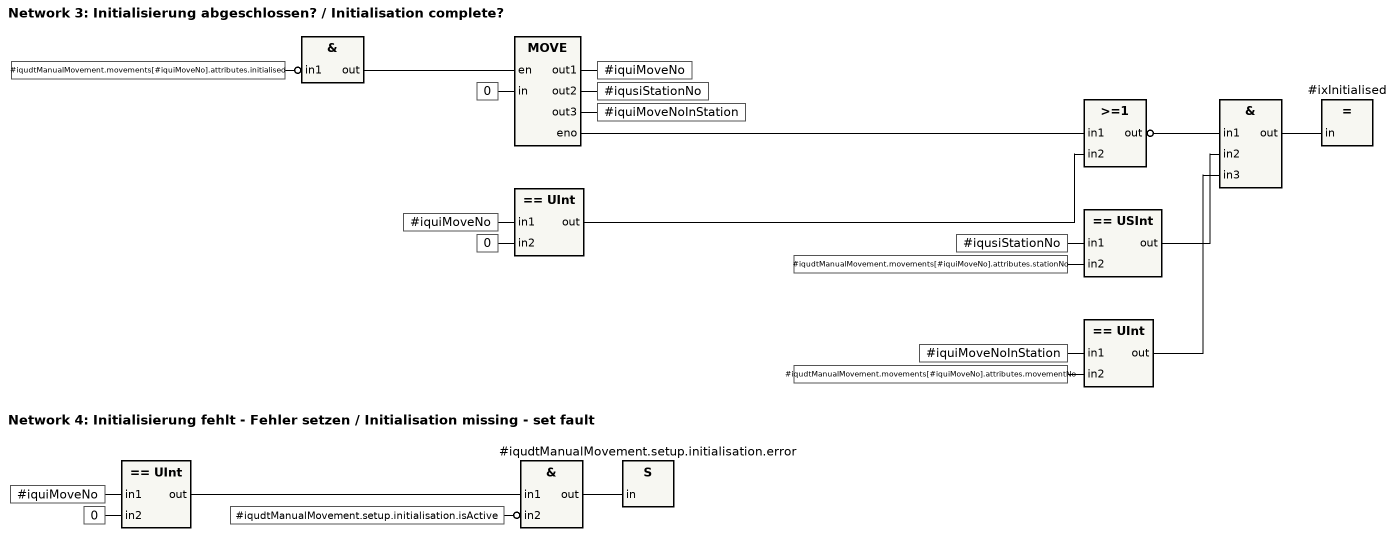
   #_w1 := NOT #iqudtManualMovement.movements[#iquiMoveNo].attributes.initialised;
   IF #_w1 THEN
       #iquiMoveNo := 0;
       #iqusiStationNo := 0;
       #iquiMoveNoInStation := 0;
   END_IF;
   #ixInitialised := NOT (#_w1 OR (#iquiMoveNo = 0)) AND (#iqusiStationNo = #iqudtManualMovement.movements[#iquiMoveNo].attributes.stationNo) AND (#iquiMoveNoInStation = #iqudtManualMovement.movements[#iquiMoveNo].attributes.movementNo);
END_REGION

REGION Network 4: Initialisierung fehlt - Fehler setzen / Initialisation missing - set fault
   IF (#iquiMoveNo = 0) AND NOT #iqudtManualMovement.setup.initialisation.isActive THEN
       #iqudtManualMovement.setup.initialisation.error := TRUE;
   END_IF;
END_REGION

REGION Network 5: Sichtbarkeit / Visibility
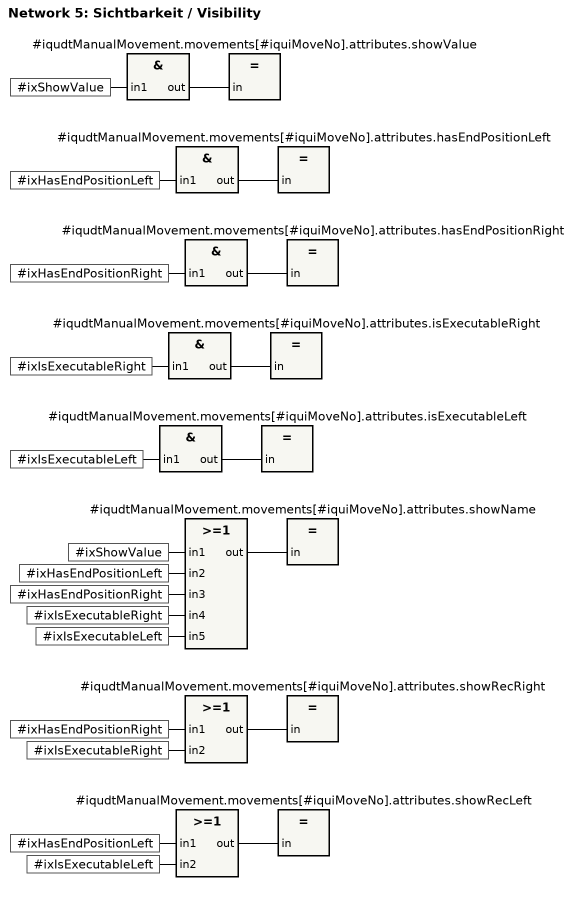
   #iqudtManualMovement.movements[#iquiMoveNo].attributes.showValue := #ixShowValue;
   #iqudtManualMovement.movements[#iquiMoveNo].attributes.hasEndPositionLeft := #ixHasEndPositionLeft;
   #iqudtManualMovement.movements[#iquiMoveNo].attributes.hasEndPositionRight := #ixHasEndPositionRight;
   #iqudtManualMovement.movements[#iquiMoveNo].attributes.isExecutableRight := #ixIsExecutableRight;
   #iqudtManualMovement.movements[#iquiMoveNo].attributes.isExecutableLeft := #ixIsExecutableLeft;
   #iqudtManualMovement.movements[#iquiMoveNo].attributes.showName := #ixShowValue OR #ixHasEndPositionLeft OR #ixHasEndPositionRight OR #ixIsExecutableRight OR #ixIsExecutableLeft;
   #iqudtManualMovement.movements[#iquiMoveNo].attributes.showRecRight := #ixHasEndPositionRight OR #ixIsExecutableRight;
   #iqudtManualMovement.movements[#iquiMoveNo].attributes.showRecLeft := #ixHasEndPositionLeft OR #ixIsExecutableLeft;
END_REGION
END_FUNCTION

FUNCTION "InitManualMovements" : Void   // FC909, SCL
{ S7_Optimized_Access := 'TRUE' }
VERSION : 0.1
   VAR_IN_OUT
      iqarudtMovements : Array[0.."SYS_MANUALMOVEMENTS"] of "typeManualMove";
   END_VAR
   VAR_TEMP
      ttusiCounter : USInt;
   END_VAR
BEGIN
   // Ersteller: Andreas Fast Automation
   // Kontakt per LinkedIn: https://www.linkedin.com/in/automation-fast-andreas/
   //
   // Projekt dient zu Demonstrationszwecken und frei genutzt werden.
   //
   // Bausteinbeschreibung:
   // 


   FOR #ttusiCounter := 0 TO "SYS_MANUALMOVEMENTS" DO
       // Initialise all manual movements
       #iqarudtMovements[#ttusiCounter].attributes.initialised := false;
       "ManualMovements".movements[#ttusiCounter].attributes.showValue := false;
       "ManualMovements".movements[#ttusiCounter].attributes.showName := false;
       "ManualMovements".movements[#ttusiCounter].attributes.showRecRight := false;
       "ManualMovements".movements[#ttusiCounter].attributes.showRecLeft := false;
       "ManualMovements".movements[#ttusiCounter].attributes.isExecutableRight := false;
       "ManualMovements".movements[#ttusiCounter].attributes.isExecutableLeft := false;
       "ManualMovements".movements[#ttusiCounter].attributes.hasEndPositionRight := false;
       "ManualMovements".movements[#ttusiCounter].attributes.hasEndPositionLeft := false;

       #iqarudtMovements[#ttusiCounter].attributes.stationNo := 0;
       #iqarudtMovements[#ttusiCounter].attributes.movementNo := 0;
   END_FOR;
END_FUNCTION

// folder: 9. Library/9.1 Framework Functions/09_Diagnosis

FUNCTION_BLOCK "StationState"   // FB9002, SCL
{ S7_Optimized_Access := 'TRUE' }
VERSION : 0.1
   VAR_INPUT
      ixIdle : Bool;   // Station wird im aktuellen Produktionsablauf nicht benötigt / Station not required in current production sequence
      ixWaitForOperator : Bool;   // Station wartet auf eine Bedieneraktion / Station waiting for operator action
      ixStarved : Bool;   // Station wartet auf Bereitstellung durch vorgelagerten Prozess / Station waiting for supply from upstream process
      ixBlocked : Bool;   // Station kann wegen nachgelagertem Prozess nicht weiterarbeiten / Station cannot continue due to downstream process
   END_VAR
   VAR_IN_OUT
      iqudtStation : "typeStation";
   END_VAR
   VAR CONSTANT
      PROCESSING : USInt := 0;   // Aktive Bearbeitung / Active processing
      FAULT : USInt := 1;   // Störung / Fault
      IDLE : USInt := 2;   // Nicht benötigt / Not required
      NOT_IN_PRODUCTION : USInt := 3;   // Nicht in Produktion / Not in production
      WAIT_FOR_OPERATOR : USInt := 4;   // Wartet auf Bediener / Waiting for operator
      BLOCKED : USInt := 5;   // Ausgabe blockiert / Output blocked
      STARVED : USInt := 6;   // Wartet auf Eingabe / Waiting for infeed
   END_VAR
BEGIN
   // Ersteller: Andreas Fast Automation
   // E-Mail: automation@fast-andreas.de
   //
   // Projekt dient zu Demonstrationszwecken und frei genutzt werden.
   //
   // Bausteinbeschreibung:
   // 
   // Priority:
   // 1. Fault
   // 2. Idle
   // 3. NotInProduction
   // 4. WaitForOperator
   // 5. Blocked
   // 6. Starved
   // 7. Processing



   IF #iqudtStation.udtSignals.isInError THEN
          #iqudtStation.usiState := #FAULT;

      ELSIF #ixIdle THEN
          #iqudtStation.usiState := #IDLE;

      ELSIF NOT #iqudtStation.udtSignals.modeAuto
          OR NOT #iqudtStation.udtSignals.releaseCycle
      THEN
          #iqudtStation.usiState := #NOT_IN_PRODUCTION;

      ELSIF #ixWaitForOperator THEN
          #iqudtStation.usiState := #WAIT_FOR_OPERATOR;

      ELSIF #ixBlocked THEN
          #iqudtStation.usiState := #BLOCKED;

      ELSIF #ixStarved THEN
          #iqudtStation.usiState := #STARVED;

      ELSE
          #iqudtStation.usiState := #PROCESSING;

      END_IF;
END_FUNCTION_BLOCK

FUNCTION_BLOCK "AlarmHandler"   // FB9009, SCL
{ S7_Optimized_Access := 'TRUE' }
VERSION : 0.1
   VAR_INPUT
      ixAck : Bool;   // Quittierung / Acknowledgement
      iiCountErrWords : Int := 4;   // Anzahl Fehlermelde-Wörter / Number of fault message words
      iiCountMessWords : Int;
   END_VAR
   VAR_OUTPUT
      qxMessage : Bool;
      qxError : Bool;   // Mindestens ein Fehler steht an / At least one fault present
   END_VAR
   VAR_IN_OUT
      iqudtAlarmsPlc : "typePlcErrMsg";
      iqudtAlarmsHmi : "typeHmiErrMsg";
   END_VAR
   VAR
      sxRisAck : Bool;
      sinstRisTrigger : R_TRIG;
      sinstTpAck : TP_TIME;
   END_VAR
   VAR_TEMP
      txAckPulse : Bool;
      tiI : Int;
      tiX : Int;
      tiLengthPlcErrors : Int;
      tiLengthPlcMessages : Int;
   END_VAR
BEGIN
   // Ersteller: Andreas Fast Automation
   // E-Mail: automation@fast-andreas.de
   //
   // Projekt dient zu Demonstrationszwecken und frei genutzt werden.
   //
   // Bausteinbeschreibung:
   // 

   // Init values
   #tiLengthPlcErrors := #iiCountErrWords * 16;
   #tiLengthPlcMessages := #iiCountMessWords * 16;

   #sinstRisTrigger(CLK := #ixAck,
                   Q => #sxRisAck);


   #sinstTpAck(IN:=#sxRisAck,
              PT:=t#1s,
              Q=>#txAckPulse);

   // Acknowledge signals for HMI
   FOR #tiI := 1 TO #iiCountErrWords DO
       IF #txAckPulse THEN
           #iqudtAlarmsHmi.alarmAckPlc[#tiI + #iiCountErrWords] := 16#FFFF;
       ELSE
           #iqudtAlarmsHmi.alarmAckPlc[#tiI + #iiCountErrWords] := 16#0;
       END_IF;
   END_FOR;


   // Clear errors of PLC
   IF #sxRisAck THEN
       FOR #tiI := 1 TO #tiLengthPlcErrors DO
           #iqudtAlarmsPlc.alarms.errorNo[#tiI] := FALSE;
       END_FOR;
   END_IF;

   // Assign plc alarms to HMI triggers
   FOR #tiI := 1 TO #iiCountErrWords DO
       #tiX := (#tiI - 1) * 16;

       #iqudtAlarmsHmi.alarmAckPlc[#tiI].%X0 := #iqudtAlarmsPlc.alarms.errorNo[#tiX + 1];
       #iqudtAlarmsHmi.alarmAckPlc[#tiI].%X1 := #iqudtAlarmsPlc.alarms.errorNo[#tiX + 2];
       #iqudtAlarmsHmi.alarmAckPlc[#tiI].%X2 := #iqudtAlarmsPlc.alarms.errorNo[#tiX + 3];
       #iqudtAlarmsHmi.alarmAckPlc[#tiI].%X3 := #iqudtAlarmsPlc.alarms.errorNo[#tiX + 4];
       #iqudtAlarmsHmi.alarmAckPlc[#tiI].%X4 := #iqudtAlarmsPlc.alarms.errorNo[#tiX + 5];
       #iqudtAlarmsHmi.alarmAckPlc[#tiI].%X5 := #iqudtAlarmsPlc.alarms.errorNo[#tiX + 6];
       #iqudtAlarmsHmi.alarmAckPlc[#tiI].%X6 := #iqudtAlarmsPlc.alarms.errorNo[#tiX + 7];
       #iqudtAlarmsHmi.alarmAckPlc[#tiI].%X7 := #iqudtAlarmsPlc.alarms.errorNo[#tiX + 8];
       #iqudtAlarmsHmi.alarmAckPlc[#tiI].%X8 := #iqudtAlarmsPlc.alarms.errorNo[#tiX + 9];
       #iqudtAlarmsHmi.alarmAckPlc[#tiI].%X9 := #iqudtAlarmsPlc.alarms.errorNo[#tiX + 10];
       #iqudtAlarmsHmi.alarmAckPlc[#tiI].%X10 := #iqudtAlarmsPlc.alarms.errorNo[#tiX + 11];
       #iqudtAlarmsHmi.alarmAckPlc[#tiI].%X11 := #iqudtAlarmsPlc.alarms.errorNo[#tiX + 12];
       #iqudtAlarmsHmi.alarmAckPlc[#tiI].%X12 := #iqudtAlarmsPlc.alarms.errorNo[#tiX + 13];
       #iqudtAlarmsHmi.alarmAckPlc[#tiI].%X13 := #iqudtAlarmsPlc.alarms.errorNo[#tiX + 14];
       #iqudtAlarmsHmi.alarmAckPlc[#tiI].%X14 := #iqudtAlarmsPlc.alarms.errorNo[#tiX + 15];
       #iqudtAlarmsHmi.alarmAckPlc[#tiI].%X15 := #iqudtAlarmsPlc.alarms.errorNo[#tiX + 16];
   END_FOR;

   // Assign PLC messages to HMI messages
   FOR #tiI := 1 TO #iiCountMessWords DO
       #tiX := (#tiI - 1) * 16;

       #iqudtAlarmsHmi.message[#tiI].%X0 := #iqudtAlarmsPlc.messages.msgNo[#tiX + 1];
       #iqudtAlarmsHmi.message[#tiI].%X1 := #iqudtAlarmsPlc.messages.msgNo[#tiX + 2];
       #iqudtAlarmsHmi.message[#tiI].%X2 := #iqudtAlarmsPlc.messages.msgNo[#tiX + 3];
       #iqudtAlarmsHmi.message[#tiI].%X3 := #iqudtAlarmsPlc.messages.msgNo[#tiX + 4];
       #iqudtAlarmsHmi.message[#tiI].%X4 := #iqudtAlarmsPlc.messages.msgNo[#tiX + 5];
       #iqudtAlarmsHmi.message[#tiI].%X5 := #iqudtAlarmsPlc.messages.msgNo[#tiX + 6];
       #iqudtAlarmsHmi.message[#tiI].%X6 := #iqudtAlarmsPlc.messages.msgNo[#tiX + 7];
       #iqudtAlarmsHmi.message[#tiI].%X7 := #iqudtAlarmsPlc.messages.msgNo[#tiX + 8];
       #iqudtAlarmsHmi.message[#tiI].%X8 := #iqudtAlarmsPlc.messages.msgNo[#tiX + 9];
       #iqudtAlarmsHmi.message[#tiI].%X9 := #iqudtAlarmsPlc.messages.msgNo[#tiX + 10];
       #iqudtAlarmsHmi.message[#tiI].%X10 := #iqudtAlarmsPlc.messages.msgNo[#tiX + 11];
       #iqudtAlarmsHmi.message[#tiI].%X11 := #iqudtAlarmsPlc.messages.msgNo[#tiX + 12];
       #iqudtAlarmsHmi.message[#tiI].%X12 := #iqudtAlarmsPlc.messages.msgNo[#tiX + 13];
       #iqudtAlarmsHmi.message[#tiI].%X13 := #iqudtAlarmsPlc.messages.msgNo[#tiX + 14];
       #iqudtAlarmsHmi.message[#tiI].%X14 := #iqudtAlarmsPlc.messages.msgNo[#tiX + 15];
       #iqudtAlarmsHmi.message[#tiI].%X15 := #iqudtAlarmsPlc.messages.msgNo[#tiX + 16];
   END_FOR;



   // set error 
   #qxError := false;
   FOR #tiI := 1 TO #tiLengthPlcErrors DO
       IF #iqudtAlarmsPlc.alarms.errorNo[#tiI] THEN
           #qxError:= TRUE;
           EXIT;
       END_IF;
   END_FOR;


   // set message
   #qxMessage := false;
   FOR #tiI := 1 TO #tiLengthPlcMessages DO
       IF #iqudtAlarmsPlc.messages.msgNo[#tiI] THEN
           #qxMessage := TRUE;
           EXIT;
       END_IF;
   END_FOR;
END_FUNCTION_BLOCK

FUNCTION_BLOCK "StationCycleTime"   // FB9103, SCL
{ S7_Optimized_Access := 'TRUE' }
VERSION : 0.7
   VAR_INPUT
      itSetpoint : Time;   // Sollzeit der aktiven Bearbeitung; Werte kleiner oder gleich 0 deaktivieren die Prüfung / Target active processing time; values less than or equal to 0 disable the check
      ixStart : Bool;   // Positive Flanke: laufenden Zyklus speichern und neuen Zyklus starten / Rising edge: store running cycle and start new cycle
      ixBottleneck : Bool := TRUE;   // TRUE: Messbereich für die Engpassdiagnose freigeben / TRUE: Enable measurement area for bottleneck diagnosis
   END_VAR
   VAR_OUTPUT
      qxError : Bool;   // Gespeicherter Fehler: ungültiger Stationszustand; Messung läuft weiter / Latched fault: invalid station state; measurement continues
   END_VAR
   VAR_IN_OUT
      iqudtCycleTime : "typeCycleTime";   // Zustandszeiten, HMI-Anzeige und Diagnosefreigabe des Messbereichs / State times, HMI display and diagnostic enable for measurement area
      iqudtStation : "typeStation";   // Stationsdaten / Station data
   END_VAR
   VAR
      sxAckOld : Bool := FALSE;   // Quittiersignal des vorherigen Aufrufs / Acknowledgement signal from previous call
      sxError : Bool := FALSE;   // Fehlerspeicher für ungültige Stationszustände / Fault memory for invalid station states
      sxStartOld : Bool := FALSE;   // Startsignal des vorherigen Aufrufs / Start signal from previous call
      sxResetOld : Bool := FALSE;   // Resetsignal des vorherigen Aufrufs / Reset signal from previous call
      sxRunning : Bool := FALSE;   // Zykluszeitmessung läuft / Cycle time measurement running
      susiPreviousState : USInt := 0;   // Stationszustand des vergangenen Aufrufintervalls / Station state during previous call interval
      sdiPreviousTick : DInt := 0;   // CPU-Zählerstand des vorherigen Aufrufs in ms / CPU counter value from previous call in ms
   END_VAR
   VAR_TEMP
      txAckEdge : Bool;   // Positive Flanke des Quittiersignals / Rising edge of acknowledgement signal
      txStartEdge : Bool;   // Positive Flanke des Startsignals / Rising edge of start signal
      txResetEdge : Bool;   // Positive Flanke des Resetsignals / Rising edge of reset signal
      tdiCurrentTick : DInt;   // Aktueller CPU-Zählerstand in ms / Current CPU counter value in ms
      tliElapsedMs : LInt;   // Vergangene Zeit seit dem vorherigen Aufruf in ms / Elapsed time since previous call in ms
      tliRemainingMs : LInt;   // Verbleibender positiver TIME-Wertebereich in ms / Remaining positive TIME value range in ms
      ttElapsed : Time;   // Begrenzte Zeitdifferenz des Aufrufintervalls / Limited time difference of call interval
      tiState : Int;   // Index beim Kopieren und Löschen der Zustandszeiten / Index for copying and clearing state times
   END_VAR
   VAR CONSTANT
      PROCESSING : Int := 0;
      FIRST_STATE : Int := 0;
      LAST_STATE : Int := 6;
      MS_PER_SECOND : LReal := LREAL#1000.0;
      ZERO_MS : LInt := LINT#0;
      MAX_TIME_MS : LInt := LINT#2_147_483_647;
      TICK_MODULUS_MS : LInt := LINT#2_147_483_648;
      ZERO_TIME : Time := T#0MS;
   END_VAR
BEGIN

       // Author: Andreas Fast Automation
       // Email: automation@fast-andreas.de
       // This project is intended for demonstration purposes and may be used freely.
       //
       // Accumulates elapsed time by station state between start edges.
       // Call once per scan after StationState, including outside Processing.
       // Internal static measurement data must be non-retentive.
       // Reset discards the current cycle and takes priority over start.
       // xNewCycle signals a completed sample, not the first measurement start.
       // TIME_TCK excludes CPU STOP time. Values saturate at the positive TIME limit.
       // Unknown states contribute only to total time, never to Processing time.
       // State errors latch until a valid acknowledgement edge; reset does not clear them.
       // Error reporting never disables measurement, cycle publication or ENO.

       REGION Detect edges and read time
           #txAckEdge := #iqudtStation.udtSignals.ack AND NOT #sxAckOld;
           #sxAckOld := #iqudtStation.udtSignals.ack;
           #txStartEdge := #ixStart AND NOT #sxStartOld;
           #sxStartOld := #ixStart;
           #txResetEdge := #iqudtStation.udtSignals.resetCycle AND NOT #sxResetOld;
           #sxResetOld := #iqudtStation.udtSignals.resetCycle;

           #tdiCurrentTick := TIME_TO_DINT(TIME_TCK());
           #iqudtCycleTime.xExists := TRUE;
           #iqudtCycleTime.xBottleneck := #ixBottleneck;
           #iqudtCycleTime.xNewCycle := FALSE;
       END_REGION

       REGION Monitor station state
           // Detect invalid input even when no measurement is running.
           IF (USINT_TO_INT(#iqudtStation.usiState) > #LAST_STATE) THEN
               #sxError := TRUE;
               #iqudtStation.udtSignals.internError := true;
           ELSIF #txAckEdge THEN
               #sxError := FALSE;
           END_IF;
           #qxError := #sxError;

       END_REGION
       REGION Accumulate elapsed interval
           IF #sxRunning THEN
               #tliElapsedMs := DINT_TO_LINT(#tdiCurrentTick)
                   - DINT_TO_LINT(#sdiPreviousTick);

               // Correct one counter wrap between consecutive calls.
               IF #tliElapsedMs < #ZERO_MS THEN
                   #tliElapsedMs := #tliElapsedMs + #TICK_MODULUS_MS;
               END_IF;

               #tliRemainingMs := #MAX_TIME_MS
                   - DINT_TO_LINT(TIME_TO_DINT(#iqudtCycleTime.stCurrentCycle.tOverall));
               IF #tliElapsedMs > #tliRemainingMs THEN
                   #tliElapsedMs := #tliRemainingMs;
               END_IF;
               #ttElapsed := DINT_TO_TIME(LINT_TO_DINT(#tliElapsedMs));

               // The previous state owns the interval ending at this call.
               IF USINT_TO_INT(#susiPreviousState) <= #LAST_STATE THEN
                   #iqudtCycleTime.stCurrentCycle.tState[#susiPreviousState] :=
                       #iqudtCycleTime.stCurrentCycle.tState[#susiPreviousState] + #ttElapsed;
               END_IF;

               #iqudtCycleTime.stCurrentCycle.tOverall :=
                   #iqudtCycleTime.stCurrentCycle.tOverall + #ttElapsed;
           END_IF;
       END_REGION

       REGION Process cycle boundary
           IF #txResetEdge THEN
               // Leave the last completed sample unchanged.
               FOR #tiState := #FIRST_STATE TO #LAST_STATE DO
                   #iqudtCycleTime.stCurrentCycle.tState[#tiState] := #ZERO_TIME;
               END_FOR;
               #iqudtCycleTime.stCurrentCycle.tOverall := #ZERO_TIME;
               #sxRunning := FALSE;

           ELSIF #txStartEdge THEN
               IF #sxRunning THEN
                   FOR #tiState := #FIRST_STATE TO #LAST_STATE DO
                       #iqudtCycleTime.stLastCycle.tState[#tiState] :=
                           #iqudtCycleTime.stCurrentCycle.tState[#tiState];
                   END_FOR;
                   #iqudtCycleTime.stLastCycle.tOverall :=
                       #iqudtCycleTime.stCurrentCycle.tOverall;
                   #iqudtCycleTime.xNewCycle := TRUE;
               END_IF;

               FOR #tiState := #FIRST_STATE TO #LAST_STATE DO
                   #iqudtCycleTime.stCurrentCycle.tState[#tiState] := #ZERO_TIME;
               END_FOR;
               #iqudtCycleTime.stCurrentCycle.tOverall := #ZERO_TIME;
               #sxRunning := TRUE;
           END_IF;
       END_REGION

       REGION Publish HMI values
           // The PLC input owns the setpoint; the HMI member is a display value.
           #iqudtCycleTime.udtHmi.rSetpointSeconds := LREAL_TO_REAL(
               DINT_TO_LREAL(TIME_TO_DINT(#itSetpoint)) / #MS_PER_SECOND);

           // Only Processing contributes to the displayed active time.
           #iqudtCycleTime.udtHmi.rActiveTimeSeconds := LREAL_TO_REAL(
               DINT_TO_LREAL(TIME_TO_DINT(
                   #iqudtCycleTime.stLastCycle.tState[#PROCESSING])) / #MS_PER_SECOND);

           #iqudtCycleTime.udtHmi.xExceeded :=
               (#itSetpoint > #ZERO_TIME)
               AND (#iqudtCycleTime.stLastCycle.tState[#PROCESSING] > #itSetpoint);
       END_REGION

       REGION Store interval reference
           #sdiPreviousTick := #tdiCurrentTick;
           #susiPreviousState := #iqudtStation.usiState;
           ENO := TRUE;
       END_REGION
END_FUNCTION_BLOCK

// folder: 9. Library/9.2 Actors

FUNCTION_BLOCK "Actor"   // FB9200, FBD
TITLE = Aktoransteuerung / Actuator control
{ S7_Optimized_Access := 'TRUE' }
VERSION : 0.1
// Ersteller: Andreas Fast Automation
// Kontakt per LinkedIn: https://www.linkedin.com/in/automation-fast-andreas/
// 
// Das Projekt dient zu Demonstrationszwecken und kann frei genutzt werden.
// 
// Bausteinbeschreibung:
// Grundlegende Funktionssteuerung eines Aktors
// Author: Andreas Fast Automation
// Kontakt per LinkedIn: https://www.linkedin.com/in/automation-fast-andreas/
// 
// This project is intended for demonstration purposes and may be used freely.
// 
// Block description:
// Basic actuator control
   VAR_INPUT
      config : USInt;   // Konfiguration Endschalterabfrage (0 = keine, 1 nur GS, 2 = Nur AS, 3 = Beide) / Limit switch feedback configuration (0 = None, 1 = Home only, 2 = Working only, 3 = Both)
      "one-sided" : Bool;   // Einseitige Ansteuerung (Nur Ansteuerung zur Arbeitsstellung vorhanden, tastend) / Single-sided actuation (working position command only, momentary)
      selfLocking : Bool;   // 1 = Selbsthaltung aktiv (Steuerimpuls setzt das Ausgangssignal) / 1 = Latching active (control pulse sets output signal)
      selfLockingInSetup : Bool;   // 1 = Selbsthaltung nur im Einrichtbetrieb bei einseitiger Spule (Ausgangsansteuerung wird setzend im Einrichten) / 1 = Latching only in setup mode with a single coil (output is latched in setup mode)
      holdEndposition : Bool;   // 1 = hält Ausgangsansteuerung aufrecht, wenn Endposition erreicht wurde / 1 = Maintains output command when end position reached
      iniHomePos : Bool;   // Grundstellung erreicht / Home position reached
      iniWorkPos : Bool;   // Arbeitsstellung erreicht / Working position reached
      interlockHome : Bool := true;   // 1 = Ansteuerung Grundstellung freigegeben / 1 = Home position actuation enabled
      interlockWork : Bool := true;   // 1 = Ansteuerung Arbeitsstellung freigegeben / 1 = Working position actuation enabled
      reactionTime : Time := t#25ms;   // Endschalter Reaktionsverzögerung / Limit switch response delay
      configNoReleaseCycle : Bool := false;   // 1 = Stationsfreigabe ist zur Ansteuerung nicht notwendig / 1 = Station enable not required for actuation
   END_VAR
   VAR_OUTPUT
      manualMoveNo : UInt;   // Bewegungsnummer für Einrichtfunktion / Movement number for setup function
      homePos : Bool;
      workPos : Bool;
   END_VAR
   VAR_IN_OUT
      actor : "typeActor";
      signals : "typeStationSignals";
      manualMovement : "typeManualMovements";
   END_VAR
   VAR
      statManualHomePos : Bool;
      statManualWorkPos : Bool;
      statSetHomeAct : Bool;
      statSetWorkAct : Bool;
      statActorManualMovement : "ActorManualMovement";
      instReactionHome : TON_TIME;
      instReactionWork : TON_TIME;
   END_VAR
   VAR_TEMP
      tempSelfLocking : Bool;
      tempHomePosConfig : Bool;
      tempWorkPosConfig : Bool;
   END_VAR
BEGIN

REGION Network 1: Selbsthaltung / Latching
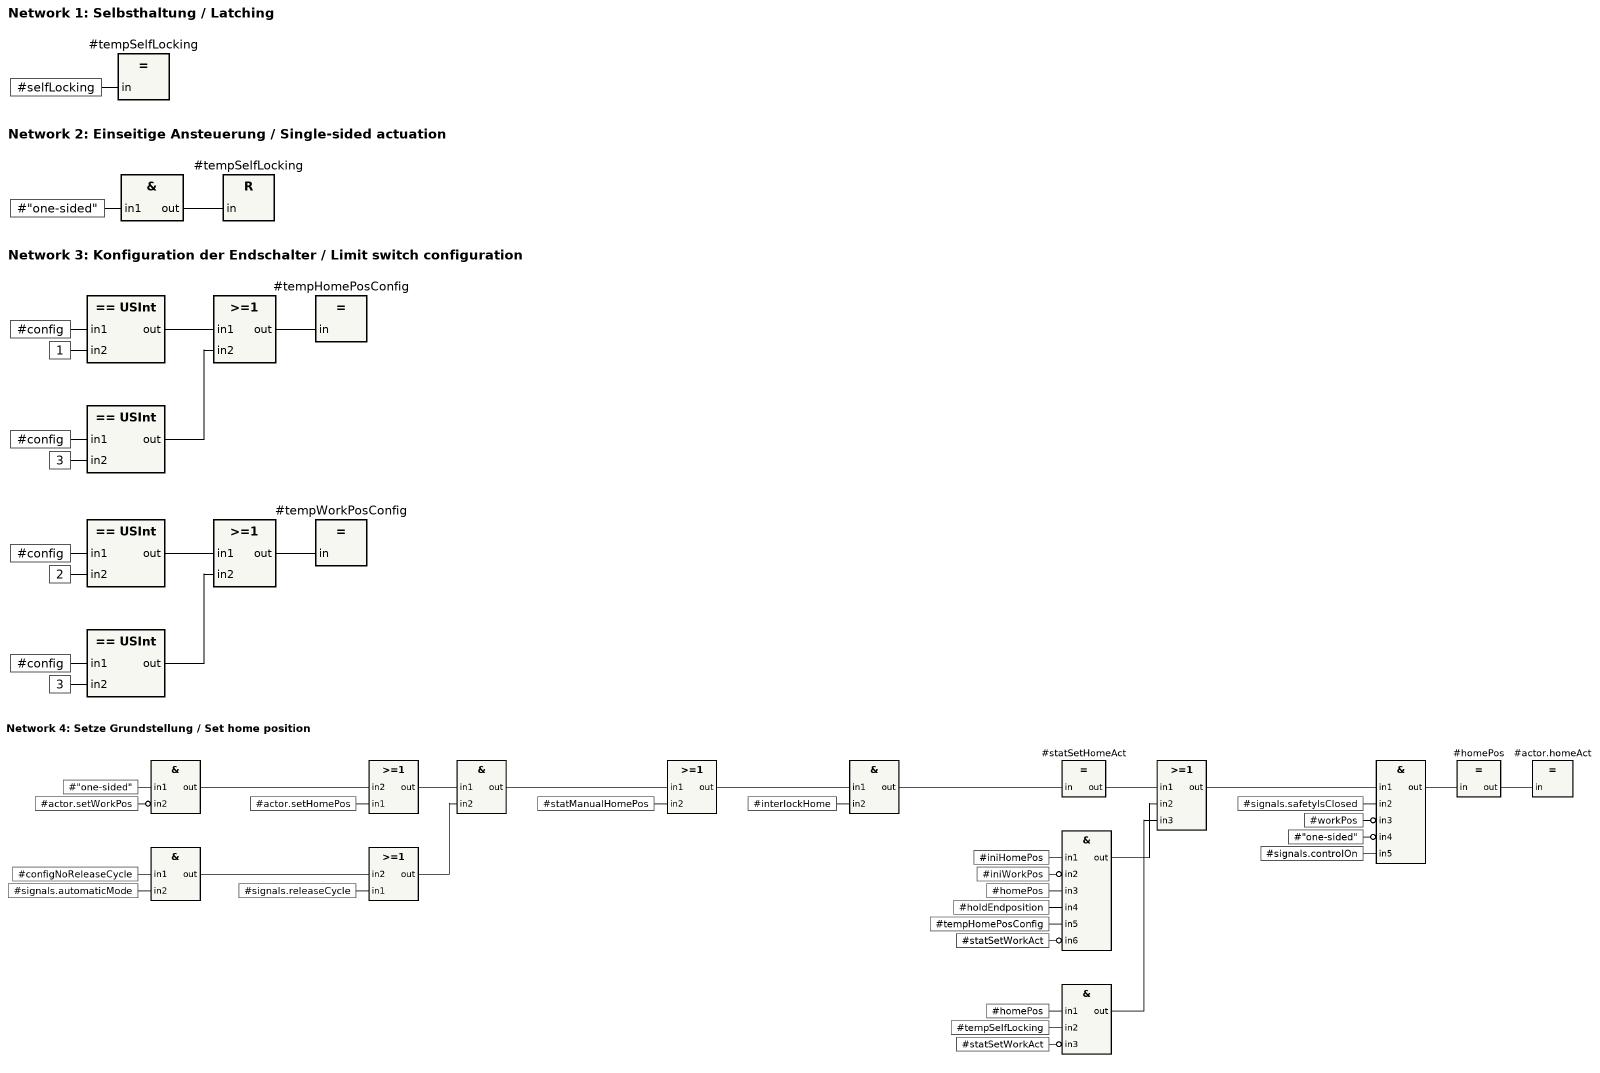
   #tempSelfLocking := #selfLocking;
END_REGION

REGION Network 2: Einseitige Ansteuerung / Single-sided actuation
   IF #"one-sided" THEN #tempSelfLocking := FALSE; END_IF;
END_REGION

REGION Network 3: Konfiguration der Endschalter / Limit switch configuration
   // 0 = Ohne Inis
   // 1 = Nur Grundstellungsabfrage
   // 2 = Nur Arbeitsstellungsabfrage
   // 3 = Beide Schaltstellungen werden abgefragt
   // 0 = No proximity sensors
   // 1 = Home position feedback only
   // 2 = Working position feedback only
   // 3 = Both end positions monitored
   #tempHomePosConfig := (#config = 1) OR (#config = 3);
   #tempWorkPosConfig := (#config = 2) OR (#config = 3);
END_REGION

REGION Network 4: Setze Grundstellung / Set home position
   #statSetHomeAct := ((((#"one-sided" AND NOT #actor.setWorkPos) OR #actor.setHomePos) AND ((#configNoReleaseCycle AND #signals.automaticMode) OR #signals.releaseCycle)) OR #statManualHomePos) AND #interlockHome;
   #homePos := (#statSetHomeAct OR (#iniHomePos AND NOT #iniWorkPos AND #homePos AND #holdEndposition AND #tempHomePosConfig AND NOT #statSetWorkAct) OR (#homePos AND #tempSelfLocking AND NOT #statSetWorkAct)) AND #signals.safetyIsClosed AND NOT #workPos AND NOT #"one-sided" AND #signals.controlOn;
   #actor.homeAct := #homePos;
END_REGION

REGION Network 5: Setze Arbeitsstellung / Set working position
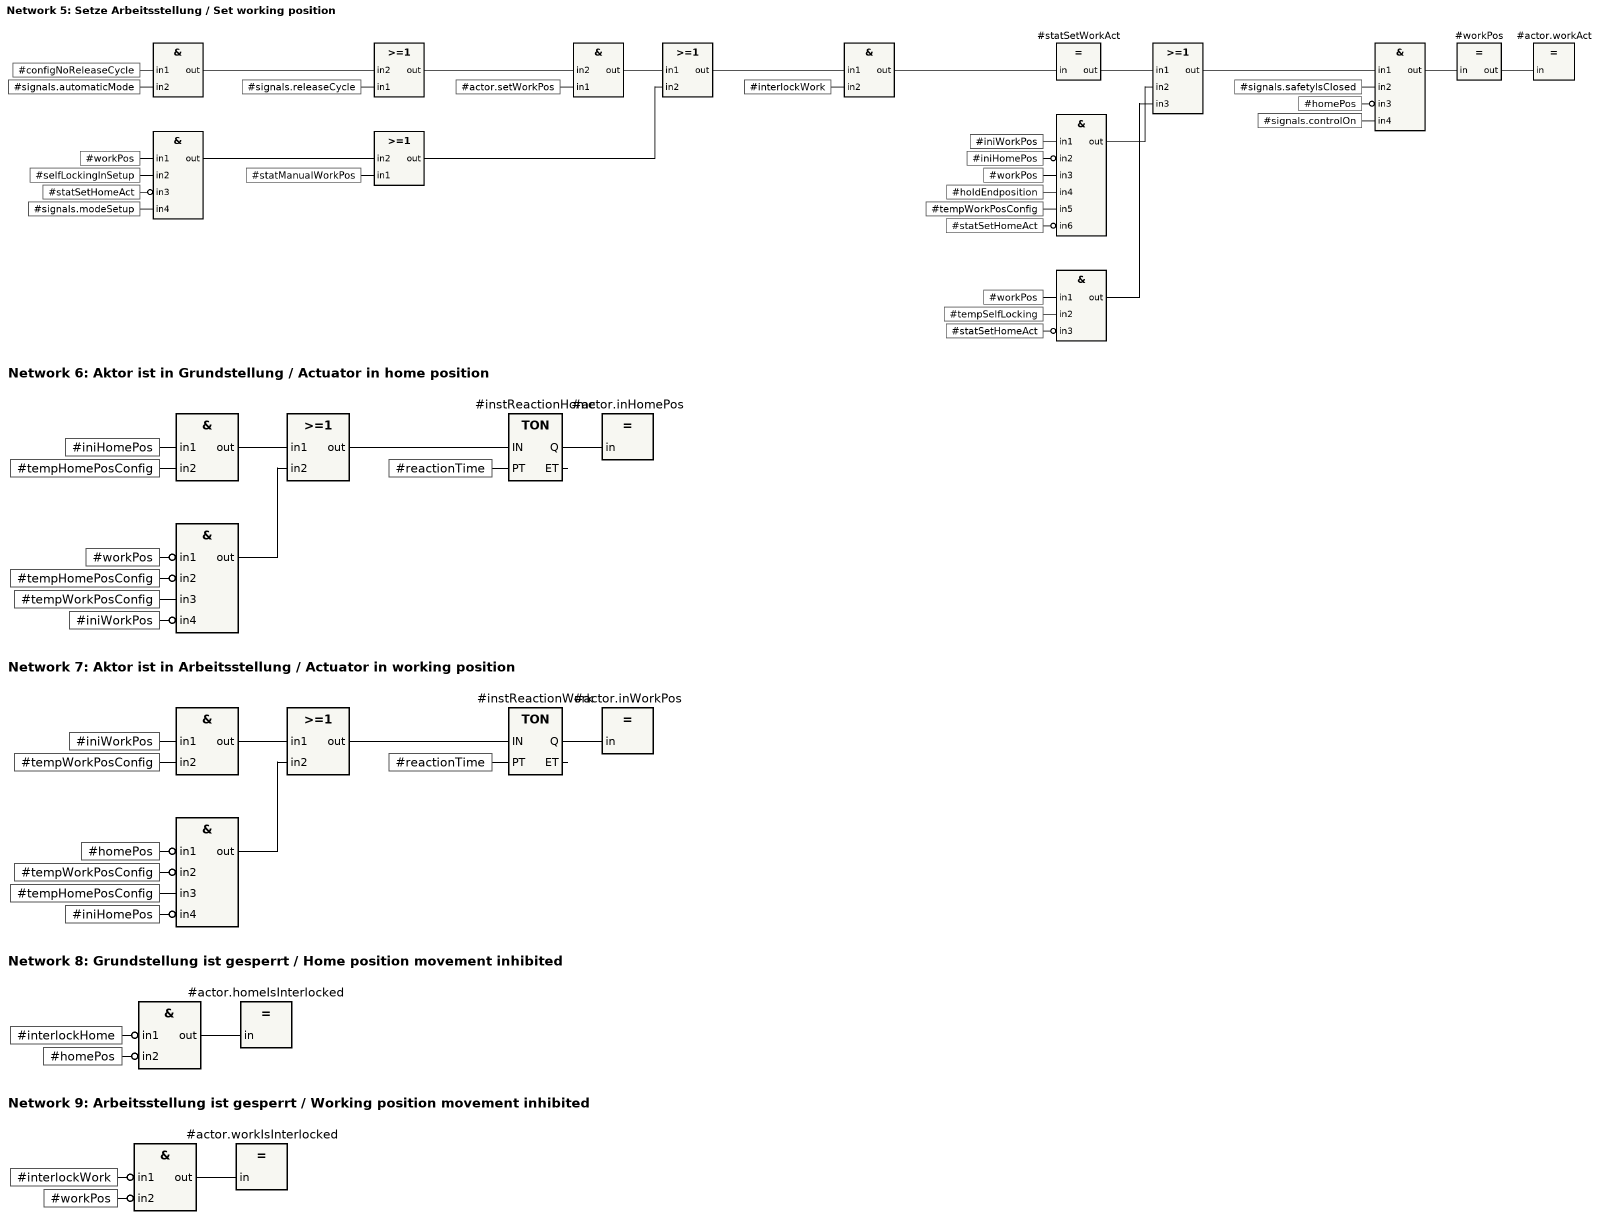
   #statSetWorkAct := ((((#configNoReleaseCycle AND #signals.automaticMode) OR #signals.releaseCycle) AND #actor.setWorkPos) OR (#workPos AND #selfLockingInSetup AND NOT #statSetHomeAct AND #signals.modeSetup) OR #statManualWorkPos) AND #interlockWork;
   #workPos := (#statSetWorkAct OR (#iniWorkPos AND NOT #iniHomePos AND #workPos AND #holdEndposition AND #tempWorkPosConfig AND NOT #statSetHomeAct) OR (#workPos AND #tempSelfLocking AND NOT #statSetHomeAct)) AND #signals.safetyIsClosed AND NOT #homePos AND #signals.controlOn;
   #actor.workAct := #workPos;
END_REGION

REGION Network 6: Aktor ist in Grundstellung / Actuator in home position
   #instReactionHome(IN := (#iniHomePos AND #tempHomePosConfig) OR (NOT #workPos AND NOT #tempHomePosConfig AND #tempWorkPosConfig AND NOT #iniWorkPos),   // TON
                     PT := #reactionTime);
   #actor.inHomePos := #instReactionHome.Q;
END_REGION

REGION Network 7: Aktor ist in Arbeitsstellung / Actuator in working position
   #instReactionWork(IN := (#iniWorkPos AND #tempWorkPosConfig) OR (NOT #homePos AND NOT #tempWorkPosConfig AND #tempHomePosConfig AND NOT #iniHomePos),   // TON
                     PT := #reactionTime);
   #actor.inWorkPos := #instReactionWork.Q;
END_REGION

REGION Network 8: Grundstellung ist gesperrt / Home position movement inhibited
   #actor.homeIsInterlocked := NOT #interlockHome AND NOT #homePos;
END_REGION

REGION Network 9: Arbeitsstellung ist gesperrt / Working position movement inhibited
   #actor.workIsInterlocked := NOT #interlockWork AND NOT #workPos;
END_REGION

REGION Network 10: Steuerung Einrichtbewegung eines Aktors / Control of an actuator setup movement
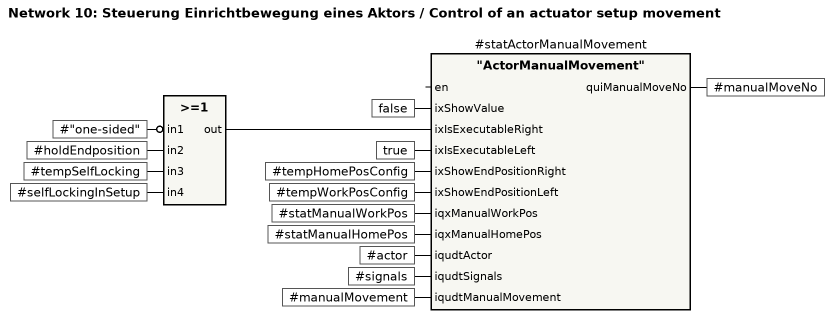
   #statActorManualMovement(ixShowValue := false,   // "ActorManualMovement"
                           ixIsExecutableRight := NOT #"one-sided" OR #holdEndposition OR #tempSelfLocking OR #selfLockingInSetup,
                           ixIsExecutableLeft := true,
                           ixShowEndPositionRight := #tempHomePosConfig,
                           ixShowEndPositionLeft := #tempWorkPosConfig,
                           iqxManualWorkPos := #statManualWorkPos,
                           iqxManualHomePos := #statManualHomePos,
                           iqudtActor := #actor,
                           iqudtSignals := #signals,
                           iqudtManualMovement := #manualMovement,
                           quiManualMoveNo => #manualMoveNo);
END_REGION
END_FUNCTION_BLOCK

FUNCTION_BLOCK "Actor_Reserved"   // FB9201, FBD
TITLE = Aktor als reservierter Platzhalter / Actuator as a reserved placeholder
{ S7_Optimized_Access := 'TRUE' }
VERSION : 0.1
// Ersteller: Andreas Fast Automation
// Kontakt per LinkedIn: https://www.linkedin.com/in/automation-fast-andreas/
// 
// Das Projekt dient zu Demonstrationszwecken und kann frei genutzt werden.
// 
// Bausteinbeschreibung:
// Author: Andreas Fast Automation
// Kontakt per LinkedIn: https://www.linkedin.com/in/automation-fast-andreas/
// 
// This project is intended for demonstration purposes and may be used freely.
// 
// Block description:
   VAR_OUTPUT
      manualMoveNo : UInt;   // Bewegungsnummer für Einrichtfunktion / Movement number for setup function
   END_VAR
   VAR_IN_OUT
      manualMovement : "typeManualMovements";
   END_VAR
   VAR
      statActorManualMovement : "ActorManualMovement";
      sudtActor : "typeActor";
      sudtSignals : "typeStationSignals";
   END_VAR
BEGIN

REGION Network 1: Steuerung Einrichtbewegung eines Aktors / Control of an actuator setup movement
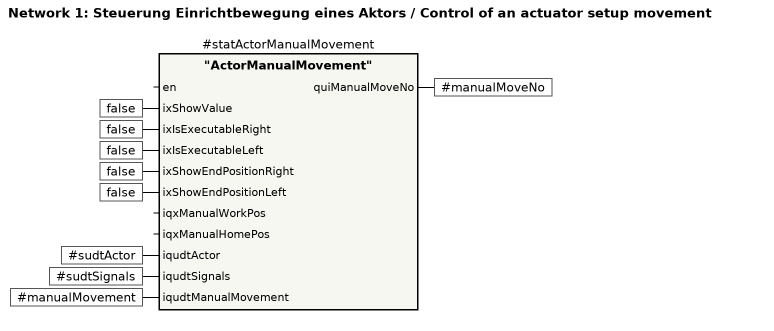
   #statActorManualMovement(ixShowValue := false,   // "ActorManualMovement"
                           ixIsExecutableRight := false,
                           ixIsExecutableLeft := false,
                           ixShowEndPositionRight := false,
                           ixShowEndPositionLeft := false,
                           iqudtActor := #sudtActor,
                           iqudtSignals := #sudtSignals,
                           iqudtManualMovement := #manualMovement,
                           quiManualMoveNo => #manualMoveNo);
END_REGION
END_FUNCTION_BLOCK

// folder: 9. Library/9.2 Actors/9.2.1 Cylinders

FUNCTION_BLOCK "Cylinder_2Out2In"   // FB9211, FBD
TITLE = Ventil: 2 Ausgänge / 2 Eingänge / Valve: 2 outputs / 2 inputs
{ S7_Optimized_Access := 'TRUE' }
VERSION : 0.1
// Ersteller: Andreas Fast Automation
// Kontakt per LinkedIn: https://www.linkedin.com/in/automation-fast-andreas/
// 
// Das Projekt dient zu Demonstrationszwecken und kann frei genutzt werden.
// 
// Bausteinbeschreibung:
// Ventilansteuerung
// Ansteuerung wird in AS/GS gehalten wenn zugehörige Endstellung vorhanden ist, selbst wenn die Aktoransteuerung rückgesetzt wird.
// Author: Andreas Fast Automation
// Kontakt per LinkedIn: https://www.linkedin.com/in/automation-fast-andreas/
// 
// This project is intended for demonstration purposes and may be used freely.
// 
// Block description:
// Valve control
// The working/home position output remains active when the corresponding end position is reached, even if the actuator command is reset.
   VAR_INPUT
      iniHomePos : Bool;   // Grundstellung erreicht / Home position reached
      iniWorkPos : Bool;   // Arbeitsstellung erreicht / Working position reached
      interlockHome : Bool := true;   // 1 = Ansteuerung Grundstellung freigegeben / 1 = Home position actuation enabled
      interlockWork : Bool := true;   // 1 = Ansteuerung Arbeitsstellung freigegeben / 1 = Working position actuation enabled
      reactionTime : Time := t#25ms;   // Endschalter Reaktionsverzögerung / Limit switch response delay
      monitoringTime : Time := T#10s;   // Überwachungszeit für Laufzeitfehler / Travel timeout monitoring time
      holdEndposition : Bool := true;   // 1 = hält Ausgangsansteuerung aufrecht, wenn Endposition erreicht wurde / 1 = Maintains output command when end position reached
   END_VAR
   VAR_OUTPUT
      manualMoveNo : UInt;   // Bewegungsnummer für Einrichtfunktion / Movement number for setup function
      homePos : Bool;
      workPos : Bool;
   END_VAR
   VAR_IN_OUT
      actor : "typeActor_2Out2In";
      signals : "typeStationSignals";
      manualMovement : "typeManualMovements";
   END_VAR
   VAR
      instActor : "Actor";
      statActor : "typeActor";
      instMonitoringHome : TON_TIME;
      instMonitoringWork : TON_TIME;
   END_VAR
BEGIN

REGION Network 1: Verbinde Aktorsignale vor Aktoransteuerung / Connect actuator signals before actuator control
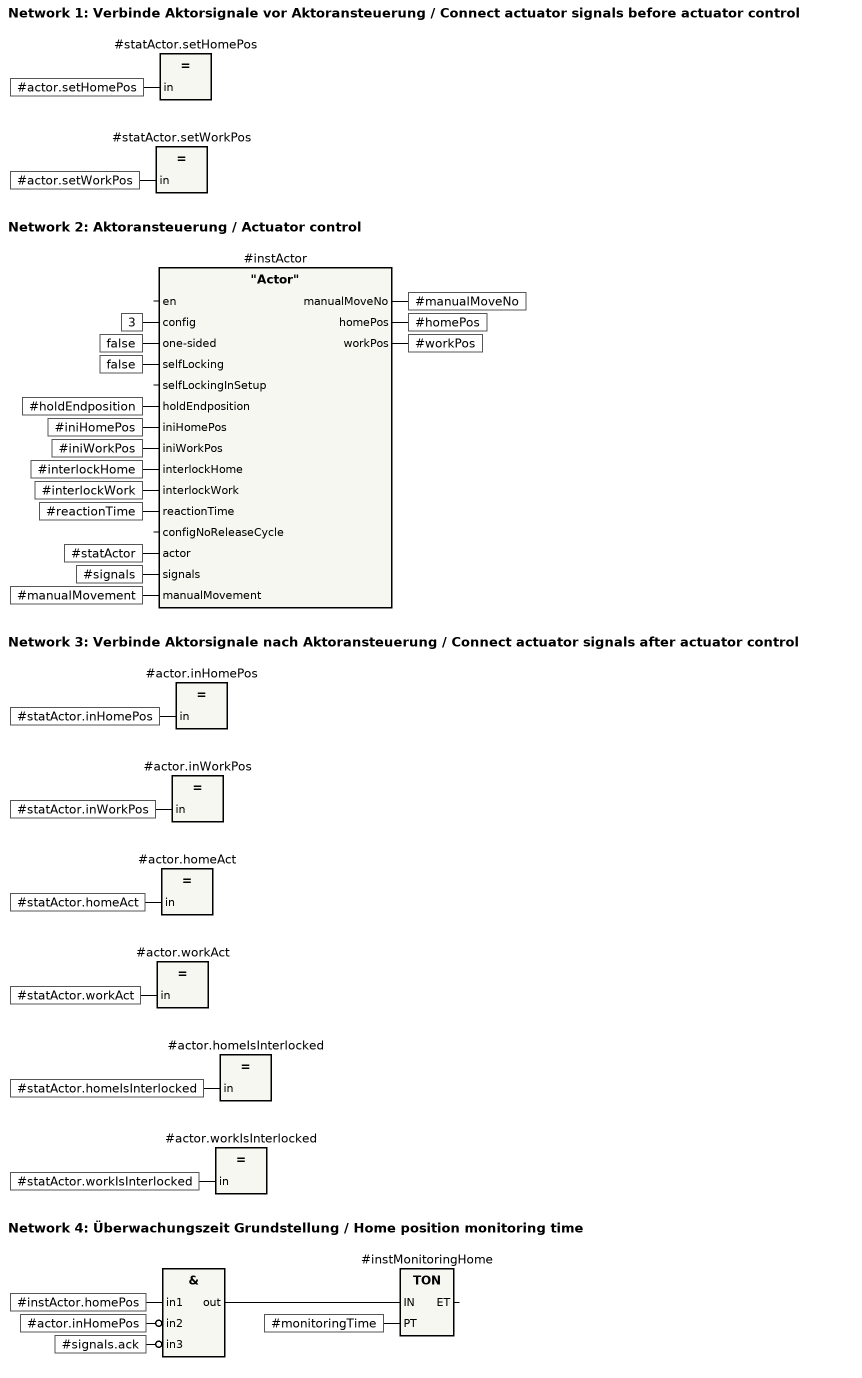
   #statActor.setHomePos := #actor.setHomePos;
   #statActor.setWorkPos := #actor.setWorkPos;
END_REGION

REGION Network 2: Aktoransteuerung / Actuator control
   #instActor(config := 3,   // "Actor"
              "one-sided" := false,
              selfLocking := false,
              holdEndposition := #holdEndposition,
              iniHomePos := #iniHomePos,
              iniWorkPos := #iniWorkPos,
              interlockHome := #interlockHome,
              interlockWork := #interlockWork,
              reactionTime := #reactionTime,
              actor := #statActor,
              signals := #signals,
              manualMovement := #manualMovement,
              manualMoveNo => #manualMoveNo,
              homePos => #homePos,
              workPos => #workPos);
END_REGION

REGION Network 3: Verbinde Aktorsignale nach Aktoransteuerung / Connect actuator signals after actuator control
   #actor.inHomePos := #statActor.inHomePos;
   #actor.inWorkPos := #statActor.inWorkPos;
   #actor.homeAct := #statActor.homeAct;
   #actor.workAct := #statActor.workAct;
   #actor.homeIsInterlocked := #statActor.homeIsInterlocked;
   #actor.workIsInterlocked := #statActor.workIsInterlocked;
END_REGION

REGION Network 4: Überwachungszeit Grundstellung / Home position monitoring time
   #instMonitoringHome(IN := #instActor.homePos AND NOT #actor.inHomePos AND NOT #signals.ack,   // TON
                       PT := #monitoringTime);
END_REGION

REGION Network 5: Überwachungszeit Arbeitsstellung / Working position monitoring time
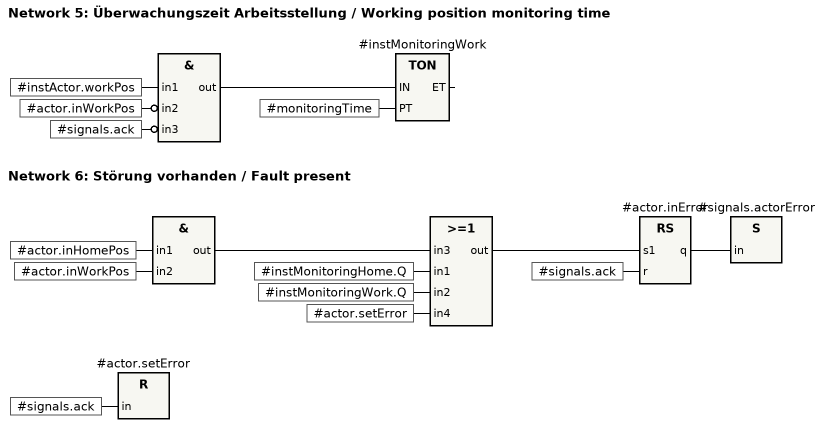
   #instMonitoringWork(IN := #instActor.workPos AND NOT #actor.inWorkPos AND NOT #signals.ack,   // TON
                       PT := #monitoringTime);
END_REGION

REGION Network 6: Störung vorhanden / Fault present
   IF #signals.ack THEN
       #actor.inError := FALSE;   // RS flip-flop
   END_IF;
   IF (#actor.inHomePos AND #actor.inWorkPos) OR #instMonitoringHome.Q OR #instMonitoringWork.Q OR #actor.setError THEN
       #actor.inError := TRUE;
   END_IF;
   IF #actor.inError THEN #signals.actorError := TRUE; END_IF;
   IF #signals.ack THEN #actor.setError := FALSE; END_IF;
END_REGION
END_FUNCTION_BLOCK

FUNCTION_BLOCK "Cylinder_1Out2In"   // FB9212, FBD
TITLE = Ventil: 1 Ausgang / 2 Eingänge / Valve: 1 output / 2 inputs
{ S7_Optimized_Access := 'TRUE' }
VERSION : 0.1
// Ersteller: Andreas Fast Automation
// Kontakt per LinkedIn: https://www.linkedin.com/in/automation-fast-andreas/
// 
// Das Projekt dient zu Demonstrationszwecken und kann frei genutzt werden.
// 
// Bausteinbeschreibung:
// Ventilansteuerung
// Ansteuerung wird in AS/GS gehalten wenn zugehörige Endstellung vorhanden ist, selbst wenn die Aktoransteuerung rückgesetzt wird.
// Author: Andreas Fast Automation
// Kontakt per LinkedIn: https://www.linkedin.com/in/automation-fast-andreas/
// 
// This project is intended for demonstration purposes and may be used freely.
// 
// Block description:
// Valve control
// The working/home position output remains active when the corresponding end position is reached, even if the actuator command is reset.
   VAR_INPUT
      iniHomePos : Bool;   // Grundstellung erreicht / Home position reached
      iniWorkPos : Bool;   // Arbeitsstellung erreicht / Working position reached
      interlockWork : Bool := true;   // 1 = Ansteuerung Arbeitsstellung freigegeben / 1 = Working position actuation enabled
      reactionTime : Time := t#25ms;   // Endschalter Reaktionsverzögerung / Limit switch response delay
      monitoringTime : Time := T#10s;   // Überwachungszeit für Laufzeitfehler / Travel timeout monitoring time
      holdEndposition : Bool := false;   // 1 = hält Ausgangsansteuerung aufrecht, wenn Endposition erreicht wurde / 1 = Maintains output command when end position reached
      configNoReleaseCycle : Bool := false;   // 1 = Stationsfreigabe ist zur Ansteuerung nicht notwendig / 1 = Station enable not required for actuation
   END_VAR
   VAR_OUTPUT
      manualMoveNo : UInt;   // Bewegungsnummer für Einrichtfunktion / Movement number for setup function
      workPos : Bool;   // SPS-Ausgang Ansteuerung Arbeitsstellung / PLC output: working position command
   END_VAR
   VAR_IN_OUT
      actor : "typeActor_1Out2In";
      signals : "typeStationSignals";
      manualMovement : "typeManualMovements";
   END_VAR
   VAR
      instActor : "Actor";
      statActor : "typeActor";
      instMonitoringHome : TON_TIME;
      instMonitoringWork : TON_TIME;
   END_VAR
BEGIN

REGION Network 1: Verbinde Aktorsignale vor Aktoransteuerung / Connect actuator signals before actuator control
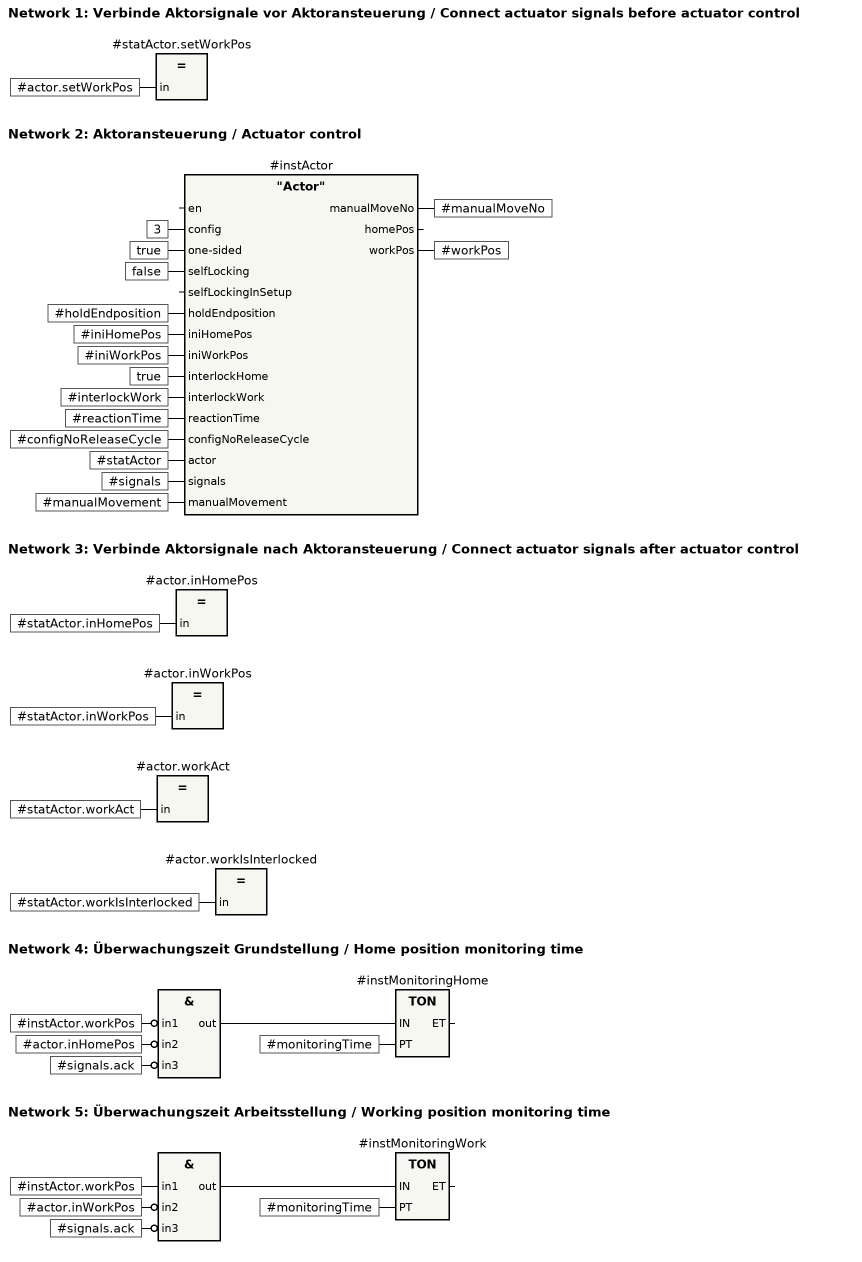
   #statActor.setWorkPos := #actor.setWorkPos;
END_REGION

REGION Network 2: Aktoransteuerung / Actuator control
   #instActor(config := 3,   // "Actor"
              "one-sided" := true,
              selfLocking := false,
              holdEndposition := #holdEndposition,
              iniHomePos := #iniHomePos,
              iniWorkPos := #iniWorkPos,
              interlockHome := true,
              interlockWork := #interlockWork,
              reactionTime := #reactionTime,
              configNoReleaseCycle := #configNoReleaseCycle,
              actor := #statActor,
              signals := #signals,
              manualMovement := #manualMovement,
              manualMoveNo => #manualMoveNo,
              workPos => #workPos);
END_REGION

REGION Network 3: Verbinde Aktorsignale nach Aktoransteuerung / Connect actuator signals after actuator control
   #actor.inHomePos := #statActor.inHomePos;
   #actor.inWorkPos := #statActor.inWorkPos;
   #actor.workAct := #statActor.workAct;
   #actor.workIsInterlocked := #statActor.workIsInterlocked;
END_REGION

REGION Network 4: Überwachungszeit Grundstellung / Home position monitoring time
   #instMonitoringHome(IN := NOT #instActor.workPos AND NOT #actor.inHomePos AND NOT #signals.ack,   // TON
                       PT := #monitoringTime);
END_REGION

REGION Network 5: Überwachungszeit Arbeitsstellung / Working position monitoring time
   #instMonitoringWork(IN := #instActor.workPos AND NOT #actor.inWorkPos AND NOT #signals.ack,   // TON
                       PT := #monitoringTime);
END_REGION

REGION Network 6: Störung vorhanden / Fault present
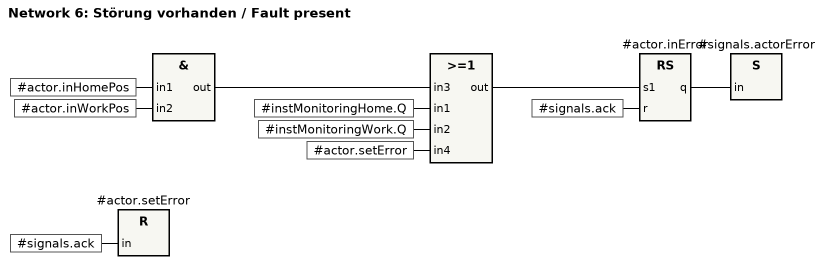
   IF #signals.ack THEN
       #actor.inError := FALSE;   // RS flip-flop
   END_IF;
   IF (#actor.inHomePos AND #actor.inWorkPos) OR #instMonitoringHome.Q OR #instMonitoringWork.Q OR #actor.setError THEN
       #actor.inError := TRUE;
   END_IF;
   IF #actor.inError THEN #signals.actorError := TRUE; END_IF;
   IF #signals.ack THEN #actor.setError := FALSE; END_IF;
END_REGION
END_FUNCTION_BLOCK

FUNCTION_BLOCK "Cylinder_2Out0In (ungetestet)"   // FB9213, FBD
TITLE = Ventil: 2 Ausgänge / 0 Eingänge / Valve: 2 outputs / 0 inputs
{ S7_Optimized_Access := 'TRUE' }
VERSION : 0.1
// Ersteller: Andreas Fast Automation
// Kontakt per LinkedIn: https://www.linkedin.com/in/automation-fast-andreas/
// 
// Das Projekt dient zu Demonstrationszwecken und kann frei genutzt werden.
// 
// Bausteinbeschreibung:
// Ventilansteuerung
// Ansteuerung wird in AS/GS gehalten wenn zugehörige Endstellung vorhanden ist, selbst wenn die Aktoransteuerung rückgesetzt wird.
// Author: Andreas Fast Automation
// Kontakt per LinkedIn: https://www.linkedin.com/in/automation-fast-andreas/
// 
// This project is intended for demonstration purposes and may be used freely.
// 
// Block description:
// Valve control
// The working/home position output remains active when the corresponding end position is reached, even if the actuator command is reset.
   VAR_INPUT
      interlockHome : Bool := true;   // 1 = Ansteuerung Grundstellung freigegeben / 1 = Home position actuation enabled
      interlockWork : Bool := true;   // 1 = Ansteuerung Arbeitsstellung freigegeben / 1 = Working position actuation enabled
      reactionTime : Time := t#25ms;   // Endschalter Reaktionsverzögerung / Limit switch response delay
      selfLockingInSetup : Bool;   // 1 = Selbsthaltung nur im Einrichtbetrieb (zweiseitige Ausgangsansteuerung setzend) / 1 = Latching only in setup mode (both directional outputs latched)
   END_VAR
   VAR_OUTPUT
      manualMoveNo : UInt;   // Bewegungsnummer für Einrichtfunktion / Movement number for setup function
      homePos : Bool;
      workPos : Bool;
   END_VAR
   VAR_IN_OUT
      actor : "typeActor_2Out0In";
      signals : "typeStationSignals";
      manualMovement : "typeManualMovements";
   END_VAR
   VAR
      instActor : "Actor";
      statActor : "typeActor";
   END_VAR
BEGIN

REGION Network 1: Verbinde Aktorsignale vor Aktoransteuerung / Connect actuator signals before actuator control
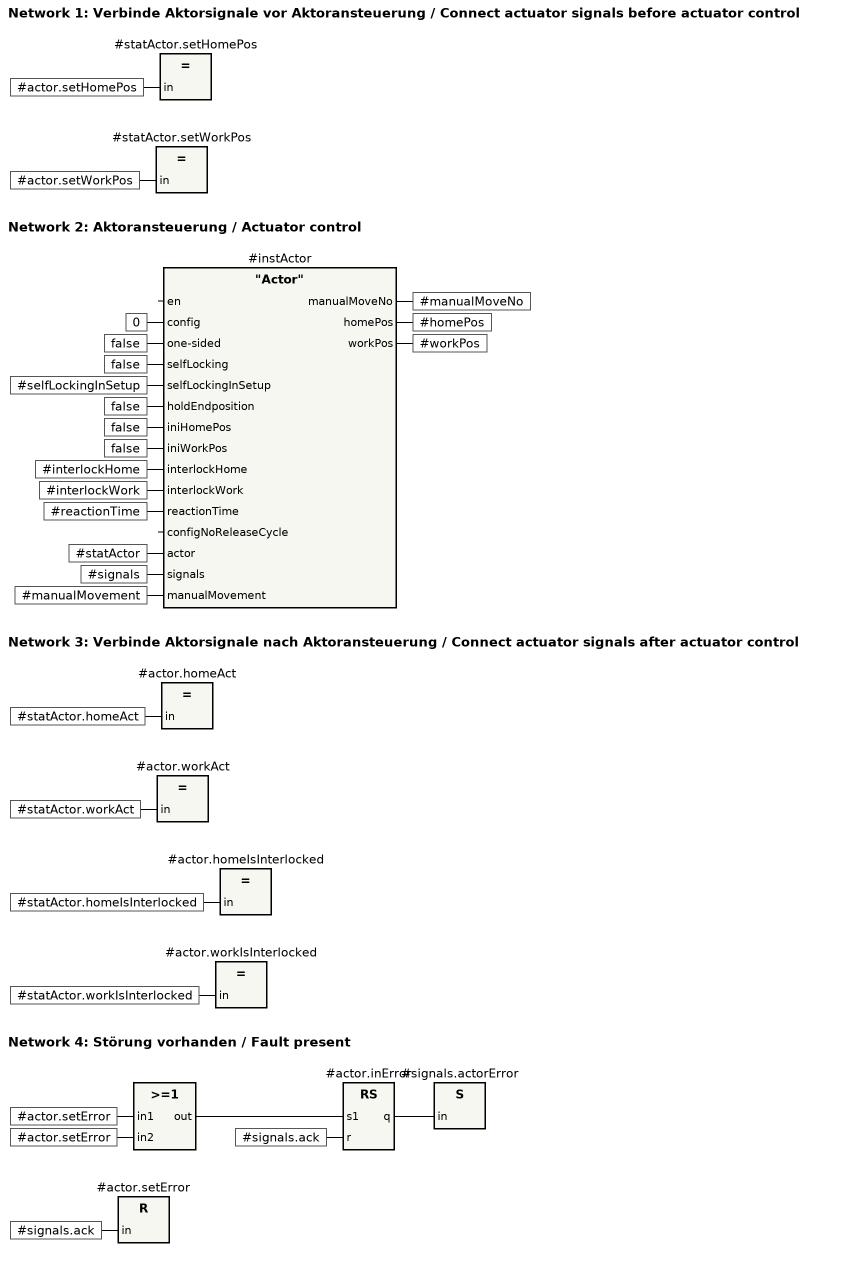
   #statActor.setHomePos := #actor.setHomePos;
   #statActor.setWorkPos := #actor.setWorkPos;
END_REGION

REGION Network 2: Aktoransteuerung / Actuator control
   #instActor(config := 0,   // "Actor"
              "one-sided" := false,
              selfLocking := false,
              selfLockingInSetup := #selfLockingInSetup,
              holdEndposition := false,
              iniHomePos := false,
              iniWorkPos := false,
              interlockHome := #interlockHome,
              interlockWork := #interlockWork,
              reactionTime := #reactionTime,
              actor := #statActor,
              signals := #signals,
              manualMovement := #manualMovement,
              manualMoveNo => #manualMoveNo,
              homePos => #homePos,
              workPos => #workPos);
END_REGION

REGION Network 3: Verbinde Aktorsignale nach Aktoransteuerung / Connect actuator signals after actuator control
   #actor.homeAct := #statActor.homeAct;
   #actor.workAct := #statActor.workAct;
   #actor.homeIsInterlocked := #statActor.homeIsInterlocked;
   #actor.workIsInterlocked := #statActor.workIsInterlocked;
END_REGION

REGION Network 4: Störung vorhanden / Fault present
   IF #signals.ack THEN
       #actor.inError := FALSE;   // RS flip-flop
   END_IF;
   IF #actor.setError OR #actor.setError THEN #actor.inError := TRUE; END_IF;
   IF #actor.inError THEN #signals.actorError := TRUE; END_IF;
   IF #signals.ack THEN #actor.setError := FALSE; END_IF;
END_REGION
END_FUNCTION_BLOCK

FUNCTION_BLOCK "Cylinder_2Out1In"   // FB9214, FBD
TITLE = Ventil: 2 Ausgänge / 1 Eingang / Valve: 2 outputs / 1 input
{ S7_Optimized_Access := 'TRUE' }
VERSION : 0.1
// Ersteller: Andreas Fast Automation
// Kontakt per LinkedIn: https://www.linkedin.com/in/automation-fast-andreas/
// 
// Das Projekt dient zu Demonstrationszwecken und kann frei genutzt werden.
// 
// Bausteinbeschreibung:
// Ventilansteuerung
// Ansteuerung wird in AS/GS gehalten wenn zugehörige Endstellung vorhanden ist, selbst wenn die Aktoransteuerung rückgesetzt wird.
// Author: Andreas Fast Automation
// Kontakt per LinkedIn: https://www.linkedin.com/in/automation-fast-andreas/
// 
// This project is intended for demonstration purposes and may be used freely.
// 
// Block description:
// Valve control
// The working/home position output remains active when the corresponding end position is reached, even if the actuator command is reset.
   VAR_INPUT
      config : Bool;   // 0 = Ini zeigt Grundstellung erreicht / 1 = Ini zeigt Arbeitsstellung erreicht / 0 = Proximity sensor indicates home position reached / 1 = Proximity sensor indicates working position reached
      iniEndPos : Bool;   // SPS-Eingang Endposition erreicht / PLC input: end position reached
      interlockHome : Bool := true;   // 1 = Ansteuerung Grundstellung freigegeben / 1 = Home position actuation enabled
      interlockWork : Bool := true;   // 1 = Ansteuerung Arbeitsstellung freigegeben / 1 = Working position actuation enabled
      reactionTime : Time := t#25ms;   // Endschalter Reaktionsverzögerung / Limit switch response delay
      monitoringTime : Time := T#10s;   // Überwachungszeit für Laufzeitfehler / Travel timeout monitoring time
      holdEndposition : Bool := false;   // 1 = hält Ausgangsansteuerung aufrecht, wenn Endposition erreicht wurde / 1 = Maintains output command when end position reached
   END_VAR
   VAR_OUTPUT
      manualMoveNo : UInt;   // Bewegungsnummer für Einrichtfunktion / Movement number for setup function
      homePos : Bool;   // SPS-Ausgang Ansteuerung Grundstellung / PLC output: home position command
      workPos : Bool;   // SPS-Ausgang Ansteuerung Arbeitsstellung / PLC output: working position command
   END_VAR
   VAR_IN_OUT
      actor : "typeActor_2Out1In";
      signals : "typeStationSignals";
      manualMovement : "typeManualMovements";
   END_VAR
   VAR
      instActor : "Actor";
      statActor : "typeActor";
      instMonitoringHome : TON_TIME;
      instMonitoringWork : TON_TIME;
   END_VAR
   VAR_TEMP
      tusiConfig : USInt;
      txInHomePos : Bool;
      txInWorkPos : Bool;
   END_VAR
BEGIN

REGION Network 1: Verbinde Aktorsignale vor Aktoransteuerung / Connect actuator signals before actuator control
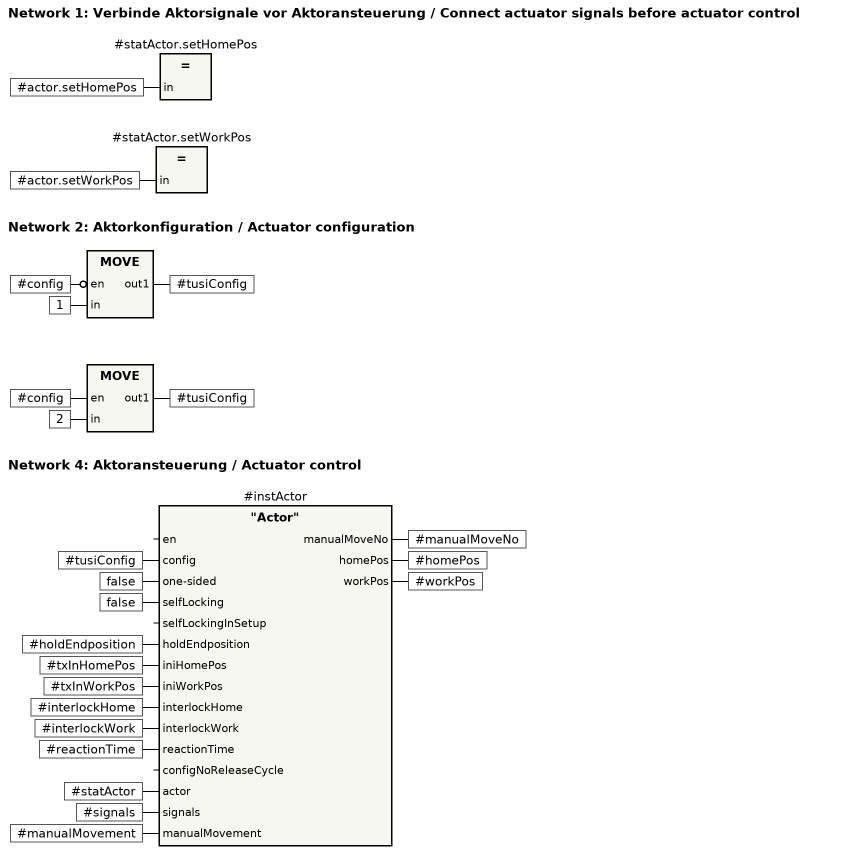
   #statActor.setHomePos := #actor.setHomePos;
   #statActor.setWorkPos := #actor.setWorkPos;
END_REGION

REGION Network 2: Aktorkonfiguration / Actuator configuration
   IF NOT #config THEN #tusiConfig := 1; END_IF;
   IF #config THEN #tusiConfig := 2; END_IF;
END_REGION

REGION Network 3 (SCL): Endschalter in Grundstellung/Arbeitsstellung / Home/working position limit switches

   IF NOT #config THEN // if sensor is checking home position
       #txInHomePos := #iniEndPos;
       #txInWorkPos := NOT #iniEndPos;

   ELSE // sensor is checking work position
       #txInWorkPos := #iniEndPos;
       #txInHomePos := NOT #iniEndPos;
   END_IF;
END_REGION

REGION Network 4: Aktoransteuerung / Actuator control
   #instActor(config := #tusiConfig,   // "Actor"
              "one-sided" := false,
              selfLocking := false,
              holdEndposition := #holdEndposition,
              iniHomePos := #txInHomePos,
              iniWorkPos := #txInWorkPos,
              interlockHome := #interlockHome,
              interlockWork := #interlockWork,
              reactionTime := #reactionTime,
              actor := #statActor,
              signals := #signals,
              manualMovement := #manualMovement,
              manualMoveNo => #manualMoveNo,
              homePos => #homePos,
              workPos => #workPos);
END_REGION

REGION Network 5: Verbinde Aktorsignale nach Aktoransteuerung / Connect actuator signals after actuator control
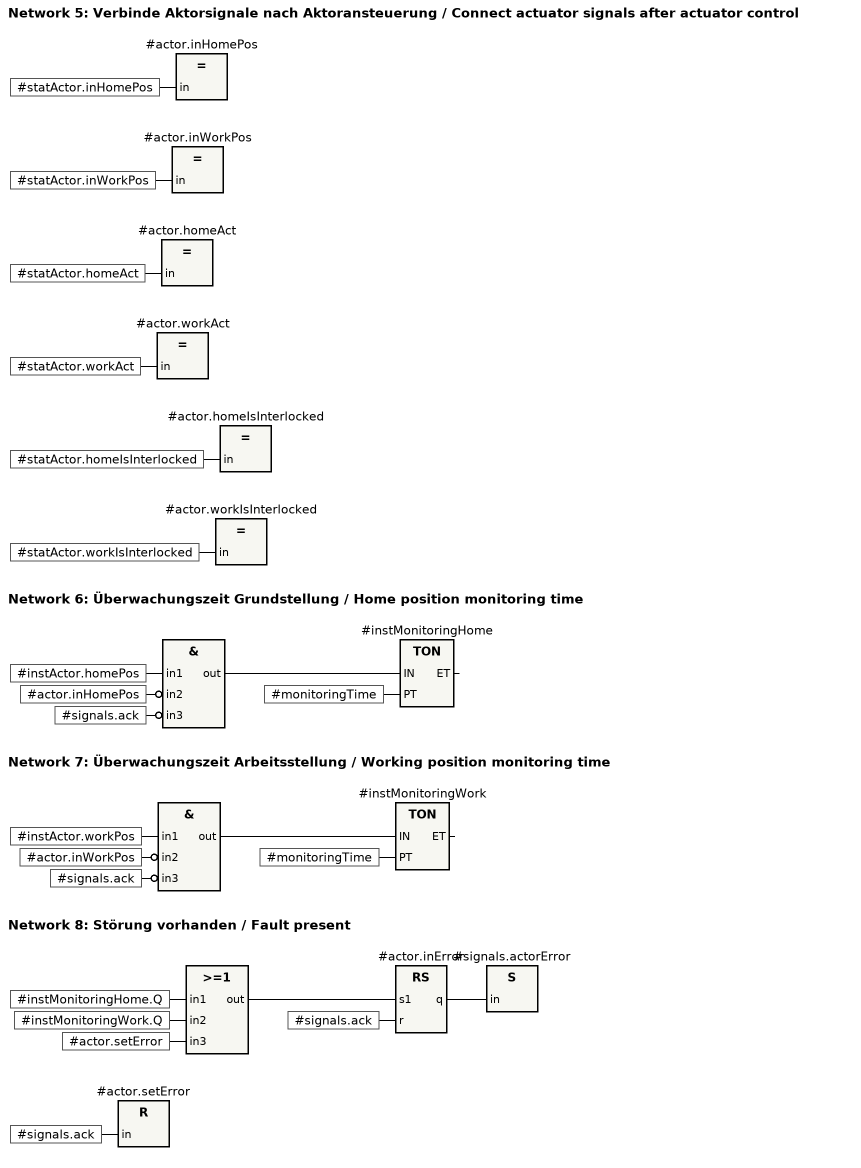
   #actor.inHomePos := #statActor.inHomePos;
   #actor.inWorkPos := #statActor.inWorkPos;
   #actor.homeAct := #statActor.homeAct;
   #actor.workAct := #statActor.workAct;
   #actor.homeIsInterlocked := #statActor.homeIsInterlocked;
   #actor.workIsInterlocked := #statActor.workIsInterlocked;
END_REGION

REGION Network 6: Überwachungszeit Grundstellung / Home position monitoring time
   #instMonitoringHome(IN := #instActor.homePos AND NOT #actor.inHomePos AND NOT #signals.ack,   // TON
                       PT := #monitoringTime);
END_REGION

REGION Network 7: Überwachungszeit Arbeitsstellung / Working position monitoring time
   #instMonitoringWork(IN := #instActor.workPos AND NOT #actor.inWorkPos AND NOT #signals.ack,   // TON
                       PT := #monitoringTime);
END_REGION

REGION Network 8: Störung vorhanden / Fault present
   IF #signals.ack THEN
       #actor.inError := FALSE;   // RS flip-flop
   END_IF;
   IF #instMonitoringHome.Q OR #instMonitoringWork.Q OR #actor.setError THEN #actor.inError := TRUE; END_IF;
   IF #actor.inError THEN #signals.actorError := TRUE; END_IF;
   IF #signals.ack THEN #actor.setError := FALSE; END_IF;
END_REGION
END_FUNCTION_BLOCK

FUNCTION_BLOCK "Cylinder_1Out1In"   // FB9215, FBD
TITLE = Ventil: 1 Ausgang / 1 Eingang / Valve: 1 output / 1 input
{ S7_Optimized_Access := 'TRUE' }
VERSION : 0.1
// Ersteller: Andreas Fast Automation
// Kontakt per LinkedIn: https://www.linkedin.com/in/automation-fast-andreas/
// 
// Das Projekt dient zu Demonstrationszwecken und kann frei genutzt werden.
// 
// Bausteinbeschreibung:
// Ventilansteuerung
// Ansteuerung wird in AS/GS gehalten wenn zugehörige Endstellung vorhanden ist, selbst wenn die Aktoransteuerung rückgesetzt wird.
// Author: Andreas Fast Automation
// Kontakt per LinkedIn: https://www.linkedin.com/in/automation-fast-andreas/
// 
// This project is intended for demonstration purposes and may be used freely.
// 
// Block description:
// Valve control
// The working/home position output remains active when the corresponding end position is reached, even if the actuator command is reset.
   VAR_INPUT
      config : Bool;   // 0 = Ini zeigt Grundstellung erreicht / 1 = Ini zeigt Arbeitsstellung erreicht / 0 = Proximity sensor indicates home position reached / 1 = Proximity sensor indicates working position reached
      iniEndPos : Bool;   // SPS-Eingang Endposition erreicht / PLC input: end position reached
      interlockWork : Bool := true;   // 1 = Ansteuerung Arbeitsstellung freigegeben / 1 = Working position actuation enabled
      reactionTime : Time := t#25ms;   // Endschalter Reaktionsverzögerung / Limit switch response delay
      monitoringTime : Time := T#10s;   // Überwachungszeit für Laufzeitfehler / Travel timeout monitoring time
      holdEndposition : Bool := false;   // 1 = hält Ausgangsansteuerung aufrecht, wenn Endposition erreicht wurde / 1 = Maintains output command when end position reached
      selfLockingInSetup : Bool;   // 1 = Selbsthaltung nur im Einrichtbetrieb (zweiseitige Ausgangsansteuerung setzend) / 1 = Latching only in setup mode (both directional outputs latched)
   END_VAR
   VAR_OUTPUT
      manualMoveNo : UInt;   // Bewegungsnummer für Einrichtfunktion / Movement number for setup function
      workPos : Bool;   // SPS-Ausgang Ansteuerung Arbeitsstellung / PLC output: working position command
   END_VAR
   VAR_IN_OUT
      actor : "typeActor_1Out1In";
      signals : "typeStationSignals";
      manualMovement : "typeManualMovements";
   END_VAR
   VAR
      instActor : "Actor";
      statActor : "typeActor";
      instMonitoringHome : TON_TIME;
      instMonitoringWork : TON_TIME;
   END_VAR
   VAR_TEMP
      tusiConfig : USInt;
      txInHomePos : Bool;
      txInWorkPos : Bool;
      txsetzendimeinrichten : Bool;
   END_VAR
BEGIN

REGION Network 1: Verbinde Aktorsignale vor Aktoransteuerung / Connect actuator signals before actuator control
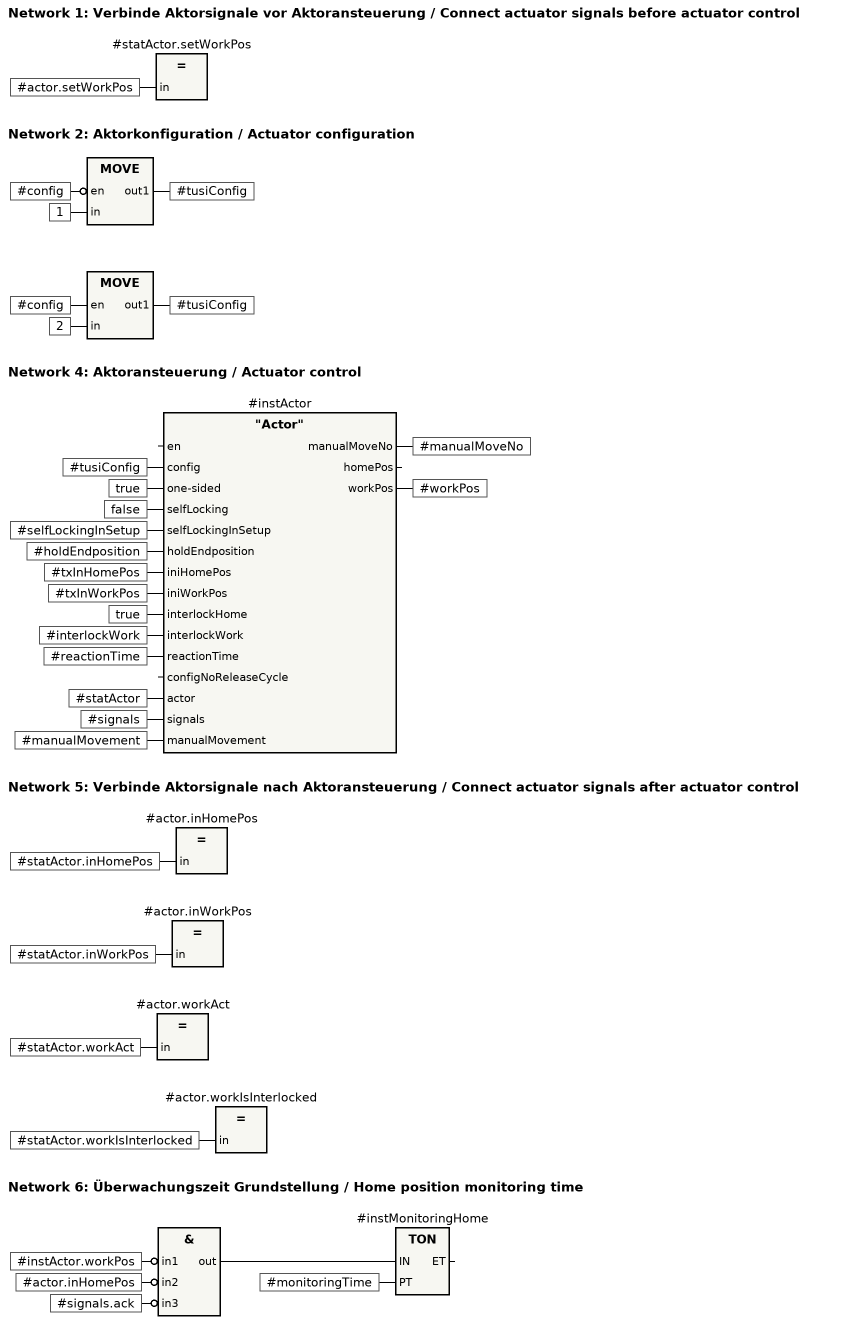
   #statActor.setWorkPos := #actor.setWorkPos;
END_REGION

REGION Network 2: Aktorkonfiguration / Actuator configuration
   IF NOT #config THEN #tusiConfig := 1; END_IF;
   IF #config THEN #tusiConfig := 2; END_IF;
END_REGION

REGION Network 3 (SCL): Endschalter in Grundstellung/Arbeitsstellung / Home/working position limit switches

   IF NOT #config THEN // if sensor is checking home position
       #txInHomePos := #iniEndPos;
       #txInWorkPos := NOT #iniEndPos;

   ELSE // sensor is checking work position
       #txInWorkPos := #iniEndPos;
       #txInHomePos := NOT #iniEndPos;
   END_IF;
END_REGION

REGION Network 4: Aktoransteuerung / Actuator control
   #instActor(config := #tusiConfig,   // "Actor"
              "one-sided" := true,
              selfLocking := false,
              selfLockingInSetup := #selfLockingInSetup,
              holdEndposition := #holdEndposition,
              iniHomePos := #txInHomePos,
              iniWorkPos := #txInWorkPos,
              interlockHome := true,
              interlockWork := #interlockWork,
              reactionTime := #reactionTime,
              actor := #statActor,
              signals := #signals,
              manualMovement := #manualMovement,
              manualMoveNo => #manualMoveNo,
              workPos => #workPos);
END_REGION

REGION Network 5: Verbinde Aktorsignale nach Aktoransteuerung / Connect actuator signals after actuator control
   #actor.inHomePos := #statActor.inHomePos;
   #actor.inWorkPos := #statActor.inWorkPos;
   #actor.workAct := #statActor.workAct;
   #actor.workIsInterlocked := #statActor.workIsInterlocked;
END_REGION

REGION Network 6: Überwachungszeit Grundstellung / Home position monitoring time
   #instMonitoringHome(IN := NOT #instActor.workPos AND NOT #actor.inHomePos AND NOT #signals.ack,   // TON
                       PT := #monitoringTime);
END_REGION

REGION Network 7: Überwachungszeit Arbeitsstellung / Working position monitoring time
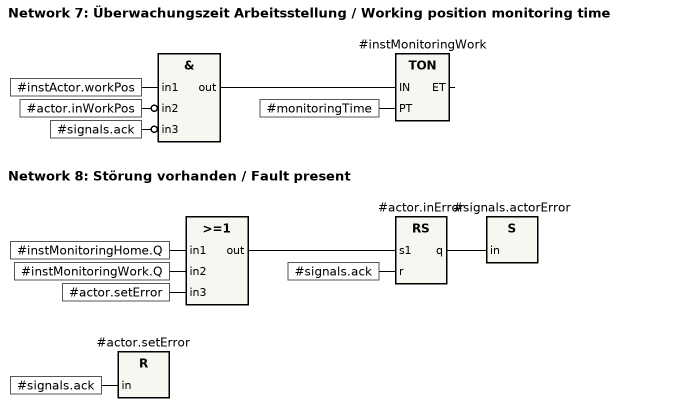
   #instMonitoringWork(IN := #instActor.workPos AND NOT #actor.inWorkPos AND NOT #signals.ack,   // TON
                       PT := #monitoringTime);
END_REGION

REGION Network 8: Störung vorhanden / Fault present
   IF #signals.ack THEN
       #actor.inError := FALSE;   // RS flip-flop
   END_IF;
   IF #instMonitoringHome.Q OR #instMonitoringWork.Q OR #actor.setError THEN #actor.inError := TRUE; END_IF;
   IF #actor.inError THEN #signals.actorError := TRUE; END_IF;
   IF #signals.ack THEN #actor.setError := FALSE; END_IF;
END_REGION
END_FUNCTION_BLOCK

FUNCTION_BLOCK "Cylinder_1Out0In"   // FB9216, FBD
TITLE = Ventil: 1 Ausgang / 0 Eingänge / Valve: 1 output / 0 inputs
{ S7_Optimized_Access := 'TRUE' }
VERSION : 0.1
// Ersteller: Andreas Fast Automation
// Kontakt per LinkedIn: https://www.linkedin.com/in/automation-fast-andreas/
// 
// Das Projekt dient zu Demonstrationszwecken und kann frei genutzt werden.
// 
// Bausteinbeschreibung:
// Ventilansteuerung
// Ansteuerung wird in AS/GS gehalten wenn zugehörige Endstellung vorhanden ist, selbst wenn die Aktoransteuerung rückgesetzt wird.
// Author: Andreas Fast Automation
// Kontakt per LinkedIn: https://www.linkedin.com/in/automation-fast-andreas/
// 
// This project is intended for demonstration purposes and may be used freely.
// 
// Block description:
// Valve control
// The working/home position output remains active when the corresponding end position is reached, even if the actuator command is reset.
   VAR_INPUT
      interlockWork : Bool := true;   // 1 = Ansteuerung Arbeitsstellung freigegeben / 1 = Working position actuation enabled
      reactionTime : Time := t#25ms;   // Endschalter Reaktionsverzögerung / Limit switch response delay
      selfLockingInSetup : Bool;   // 1 = Selbsthaltung nur im Einrichtbetrieb (zweiseitige Ausgangsansteuerung setzend) / 1 = Latching only in setup mode (both directional outputs latched)
   END_VAR
   VAR_OUTPUT
      manualMoveNo : UInt;   // Bewegungsnummer für Einrichtfunktion / Movement number for setup function
      workPos : Bool;   // SPS-Ausgang Ansteuerung Arbeitsstellung / PLC output: working position command
   END_VAR
   VAR_IN_OUT
      actor : "typeActor_1Out0In";
      signals : "typeStationSignals";
      manualMovement : "typeManualMovements";
   END_VAR
   VAR
      instActor : "Actor";
      statActor : "typeActor";
   END_VAR
BEGIN

REGION Network 1: Verbinde Aktorsignale vor Aktoransteuerung / Connect actuator signals before actuator control
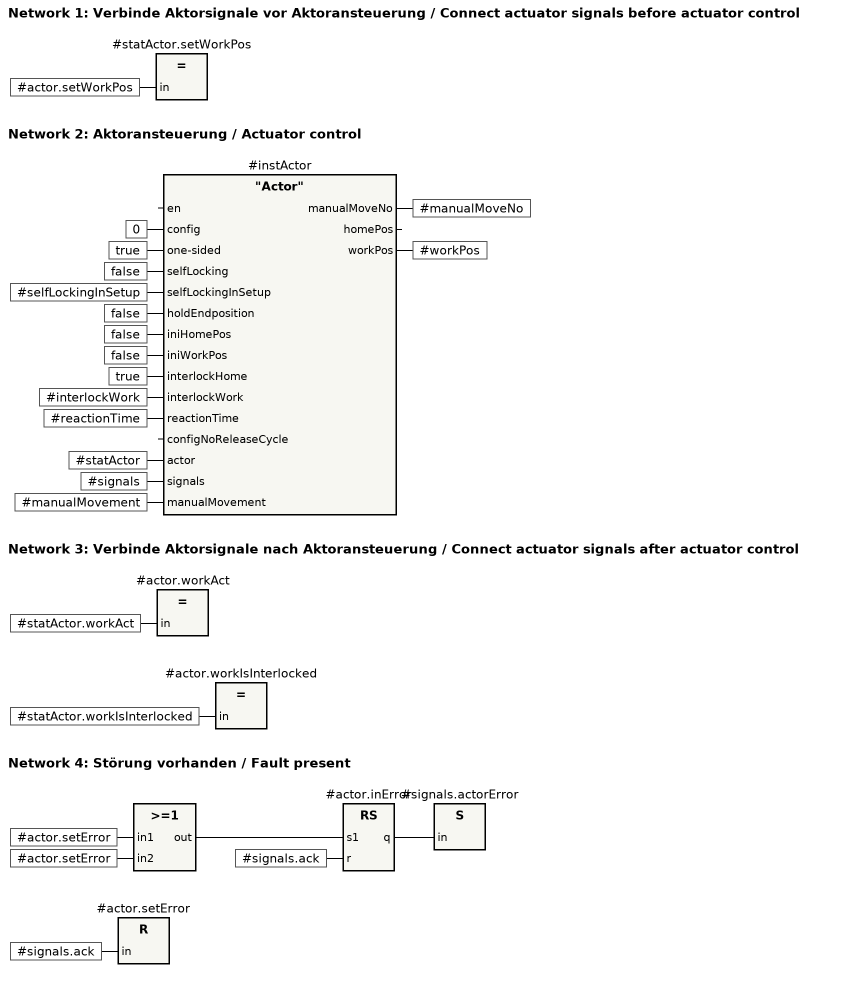
   #statActor.setWorkPos := #actor.setWorkPos;
END_REGION

REGION Network 2: Aktoransteuerung / Actuator control
   #instActor(config := 0,   // "Actor"
              "one-sided" := true,
              selfLocking := false,
              selfLockingInSetup := #selfLockingInSetup,
              holdEndposition := false,
              iniHomePos := false,
              iniWorkPos := false,
              interlockHome := true,
              interlockWork := #interlockWork,
              reactionTime := #reactionTime,
              actor := #statActor,
              signals := #signals,
              manualMovement := #manualMovement,
              manualMoveNo => #manualMoveNo,
              workPos => #workPos);
END_REGION

REGION Network 3: Verbinde Aktorsignale nach Aktoransteuerung / Connect actuator signals after actuator control
   #actor.workAct := #statActor.workAct;
   #actor.workIsInterlocked := #statActor.workIsInterlocked;
END_REGION

REGION Network 4: Störung vorhanden / Fault present
   IF #signals.ack THEN
       #actor.inError := FALSE;   // RS flip-flop
   END_IF;
   IF #actor.setError OR #actor.setError THEN #actor.inError := TRUE; END_IF;
   IF #actor.inError THEN #signals.actorError := TRUE; END_IF;
   IF #signals.ack THEN #actor.setError := FALSE; END_IF;
END_REGION
END_FUNCTION_BLOCK

// folder: 9. Library/9.2 Actors/9.2.2 Motors

FUNCTION_BLOCK "Motor_1Out"   // FB9221, FBD
TITLE = Motoransteuerung / Motor control
{ S7_Optimized_Access := 'TRUE' }
VERSION : 0.1
// Ersteller: Andreas Fast Automation
// Kontakt per LinkedIn: https://www.linkedin.com/in/automation-fast-andreas/
// 
// Das Projekt dient zu Demonstrationszwecken und kann frei genutzt werden.
// 
// Bausteinbeschreibung:
// Author: Andreas Fast Automation
// Kontakt per LinkedIn: https://www.linkedin.com/in/automation-fast-andreas/
// 
// This project is intended for demonstration purposes and may be used freely.
// 
// Block description:
   VAR_INPUT
      circuitBreaker : Bool := true;   // 1 = Schutzschalter OK / 1 = Circuit breaker OK
      interlockWork : Bool := true;   // 1 = Ansteuerung Arbeitsstellung freigegeben / 1 = Working position actuation enabled
      errorExtern : Bool;   // 1 = externer Fehler / 1 = External fault
      configNoReleaseCycle : Bool := false;   // 1 = Stationsfreigabe ist zur Ansteuerung nicht notwendig / 1 = Station enable not required for actuation
   END_VAR
   VAR_OUTPUT
      manualMoveNo : UInt;   // Bewegungsnummer für Einrichtfunktion / Movement number for setup function
      workPos : Bool;
   END_VAR
   VAR_IN_OUT
      actor : "typeActor_1Out0In";
      signals : "typeStationSignals";
      manualMovement : "typeManualMovements";
   END_VAR
   VAR
      instActor : "Actor";
      statActor : "typeActor";
   END_VAR
BEGIN

REGION Network 1: Verbinde Aktorsignale vor Aktoransteuerung / Connect actuator signals before actuator control
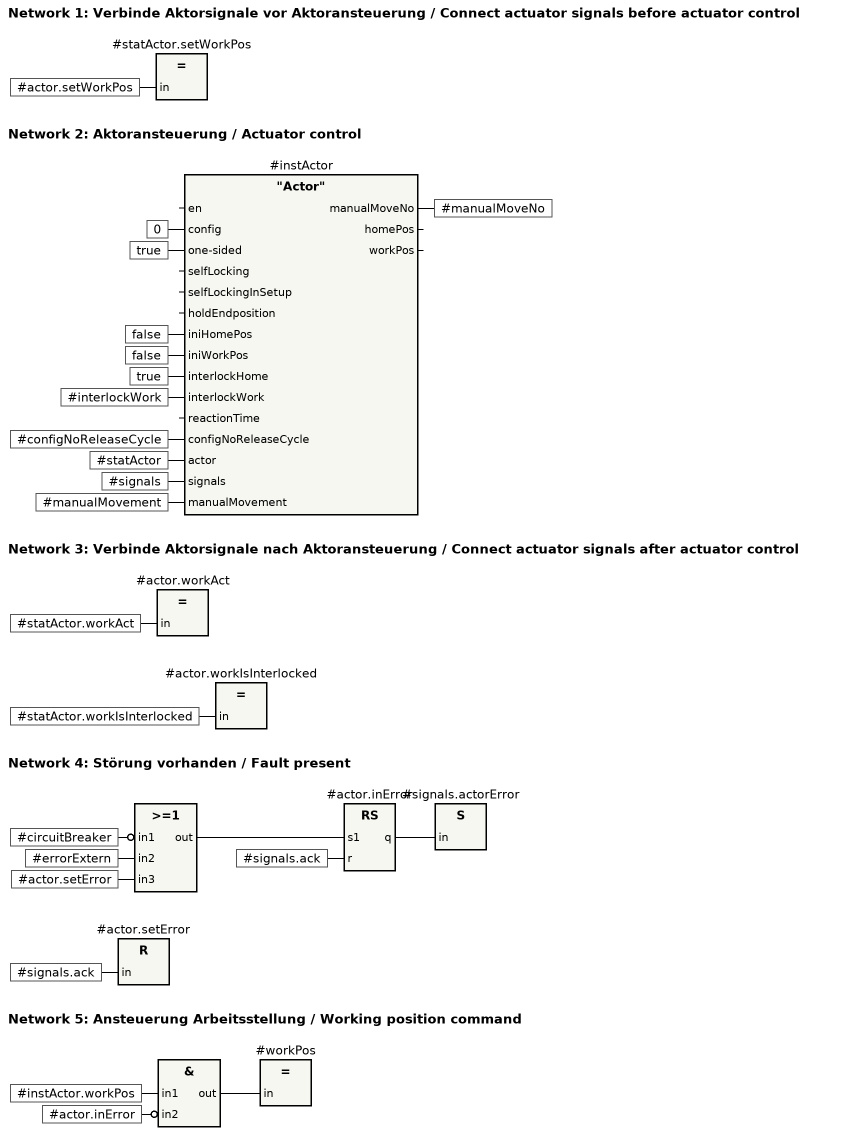
   #statActor.setWorkPos := #actor.setWorkPos;
END_REGION

REGION Network 2: Aktoransteuerung / Actuator control
   #instActor(config := 0,   // "Actor"
              "one-sided" := true,
              iniHomePos := false,
              iniWorkPos := false,
              interlockHome := true,
              interlockWork := #interlockWork,
              configNoReleaseCycle := #configNoReleaseCycle,
              actor := #statActor,
              signals := #signals,
              manualMovement := #manualMovement,
              manualMoveNo => #manualMoveNo);
END_REGION

REGION Network 3: Verbinde Aktorsignale nach Aktoransteuerung / Connect actuator signals after actuator control
   #actor.workAct := #statActor.workAct;
   #actor.workIsInterlocked := #statActor.workIsInterlocked;
END_REGION

REGION Network 4: Störung vorhanden / Fault present
   IF #signals.ack THEN
       #actor.inError := FALSE;   // RS flip-flop
   END_IF;
   IF NOT #circuitBreaker OR #errorExtern OR #actor.setError THEN #actor.inError := TRUE; END_IF;
   IF #actor.inError THEN #signals.actorError := TRUE; END_IF;
   IF #signals.ack THEN #actor.setError := FALSE; END_IF;
END_REGION

REGION Network 5: Ansteuerung Arbeitsstellung / Working position command
   #workPos := #instActor.workPos AND NOT #actor.inError;
END_REGION
END_FUNCTION_BLOCK

FUNCTION_BLOCK "Motor_2Out"   // FB9222, FBD
TITLE = Motoransteuerung / Motor control
{ S7_Optimized_Access := 'TRUE' }
VERSION : 0.1
// Ersteller: Andreas Fast Automation
// Kontakt per LinkedIn: https://www.linkedin.com/in/automation-fast-andreas/
// 
// Das Projekt dient zu Demonstrationszwecken und kann frei genutzt werden.
// 
// Bausteinbeschreibung:
// Author: Andreas Fast Automation
// Kontakt per LinkedIn: https://www.linkedin.com/in/automation-fast-andreas/
// 
// This project is intended for demonstration purposes and may be used freely.
// 
// Block description:
   VAR_INPUT
      circuitBreaker : Bool := true;   // 1 = Schutzschalter OK / 1 = Circuit breaker OK
      interlockHome : Bool := true;   // 1 = Ansteuerung Grundstellung freigegeben / 1 = Home position actuation enabled
      interlockWork : Bool := true;   // 1 = Ansteuerung Arbeitsstellung freigegeben / 1 = Working position actuation enabled
      errorExtern : Bool;   // 1 = externer Fehler / 1 = External fault
      configNoReleaseCycle : Bool := false;   // 1 = Stationsfreigabe ist zur Ansteuerung nicht notwendig / 1 = Station enable not required for actuation
   END_VAR
   VAR_OUTPUT
      manualMoveNo : UInt;   // Bewegungsnummer für Einrichtfunktion / Movement number for setup function
      homePos : Bool;
      workPos : Bool;
   END_VAR
   VAR_IN_OUT
      actor : "typeActor_2Out0In";
      signals : "typeStationSignals";
      manualMovement : "typeManualMovements";
   END_VAR
   VAR
      instActor : "Actor";
      statActor : "typeActor";
   END_VAR
BEGIN

REGION Network 1: Verbinde Aktorsignale vor Aktoransteuerung / Connect actuator signals before actuator control
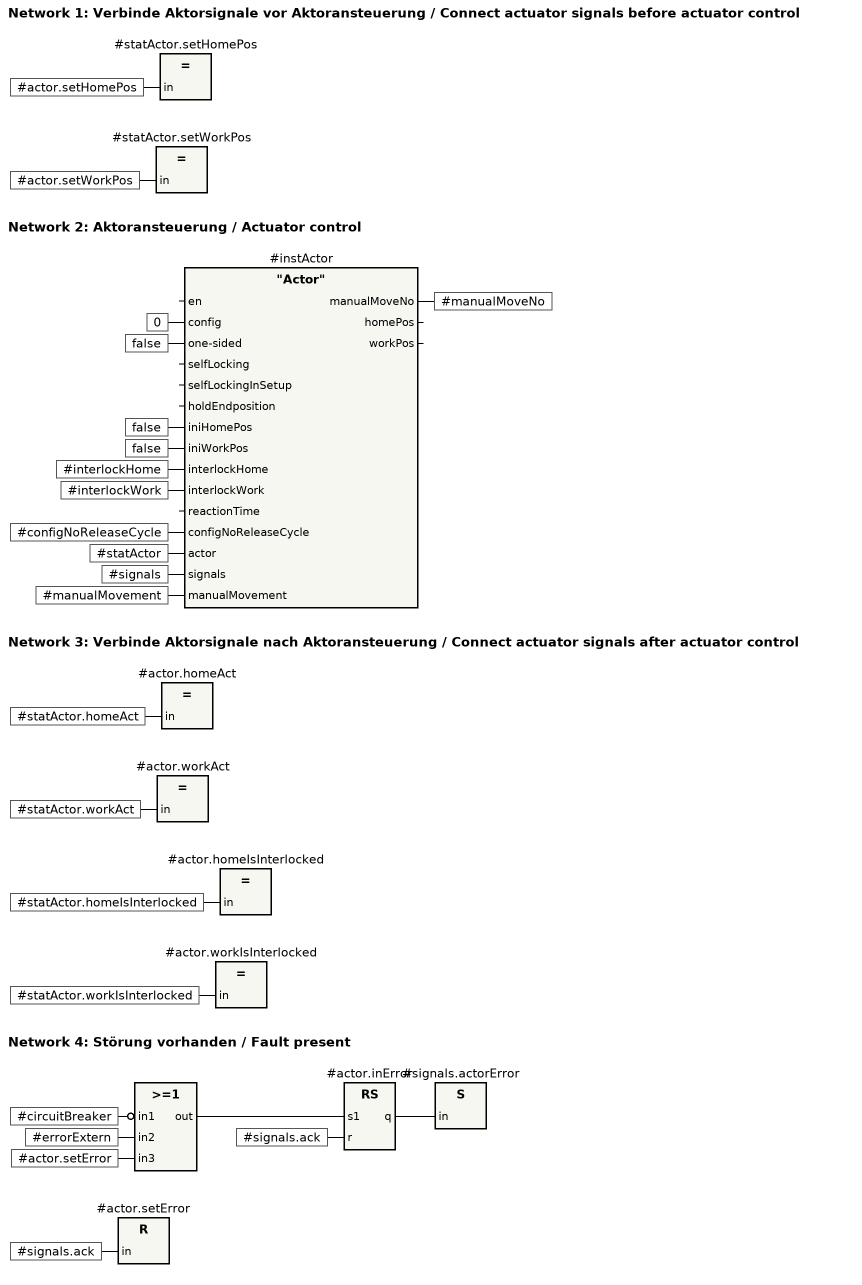
   #statActor.setHomePos := #actor.setHomePos;
   #statActor.setWorkPos := #actor.setWorkPos;
END_REGION

REGION Network 2: Aktoransteuerung / Actuator control
   #instActor(config := 0,   // "Actor"
              "one-sided" := false,
              iniHomePos := false,
              iniWorkPos := false,
              interlockHome := #interlockHome,
              interlockWork := #interlockWork,
              configNoReleaseCycle := #configNoReleaseCycle,
              actor := #statActor,
              signals := #signals,
              manualMovement := #manualMovement,
              manualMoveNo => #manualMoveNo);
END_REGION

REGION Network 3: Verbinde Aktorsignale nach Aktoransteuerung / Connect actuator signals after actuator control
   #actor.homeAct := #statActor.homeAct;
   #actor.workAct := #statActor.workAct;
   #actor.homeIsInterlocked := #statActor.homeIsInterlocked;
   #actor.workIsInterlocked := #statActor.workIsInterlocked;
END_REGION

REGION Network 4: Störung vorhanden / Fault present
   IF #signals.ack THEN
       #actor.inError := FALSE;   // RS flip-flop
   END_IF;
   IF NOT #circuitBreaker OR #errorExtern OR #actor.setError THEN #actor.inError := TRUE; END_IF;
   IF #actor.inError THEN #signals.actorError := TRUE; END_IF;
   IF #signals.ack THEN #actor.setError := FALSE; END_IF;
END_REGION

REGION Network 5: Ansteuerung Grundstellung / Home position command
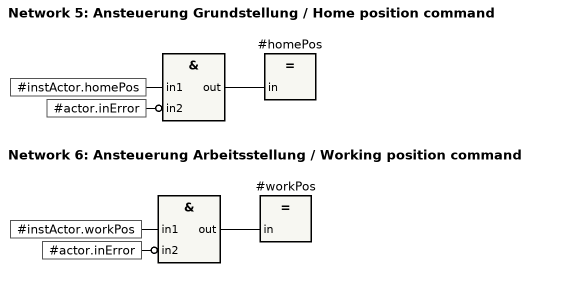
   #homePos := #instActor.homePos AND NOT #actor.inError;
END_REGION

REGION Network 6: Ansteuerung Arbeitsstellung / Working position command
   #workPos := #instActor.workPos AND NOT #actor.inError;
END_REGION
END_FUNCTION_BLOCK

// folder: 9. Library/9.2 Actors/9.2.5 Cameras

FUNCTION_BLOCK "Actor_1Out_SimpleCamera"   // FB9202, FBD
TITLE = Aktor als einfache Kamera / Actuator as a simple camera
{ S7_Optimized_Access := 'TRUE' }
VERSION : 0.1
// Ersteller: Andreas Fast Automation
// Kontakt per LinkedIn: https://www.linkedin.com/in/automation-fast-andreas/
// 
// Das Projekt dient zu Demonstrationszwecken und kann frei genutzt werden.
// 
// Bausteinbeschreibung:
// Author: Andreas Fast Automation
// Kontakt per LinkedIn: https://www.linkedin.com/in/automation-fast-andreas/
// 
// This project is intended for demonstration purposes and may be used freely.
// 
// Block description:
   VAR_INPUT
      ixReady : Bool;   // Kamera ist bereit / Camera ready
      ixBusy : Bool;   // Kamera ist aktiv / Camera active
      ixResultOk : Bool;   // Ergebnis OK / Result OK
      ixResultNok : Bool;   // Ergebnis NOK / Result NOK
      interlockWork : Bool := true;   // 1 = Ansteuerung Arbeitsstellung freigegeben / 1 = Working position actuation enabled
      configNoReleaseCycle : Bool := false;   // 1 = Stationsfreigabe ist zur Ansteuerung nicht notwendig / 1 = Station enable not required for actuation
   END_VAR
   VAR_OUTPUT
      manualMoveNo1 : UInt;   // Bewegungsnummer für Einrichtfunktion / Movement number for setup function
      manualMoveNo2 : UInt;   // Bewegungsnummer für Einrichtfunktion / Movement number for setup function
      enable : Bool;   // SPS-Ausgang Ansteuerung Kamera einschalten / PLC output: camera power-on command
      trigger : Bool;   // SPS-Ausgang Ansteuerung Kamera triggern / PLC output: camera trigger command
   END_VAR
   VAR_IN_OUT
      actor : "typeActor_1Out_SimpleCamera";
      signals : "typeStationSignals";
      manualMovement : "typeManualMovements";
   END_VAR
   VAR
      statActorManualMovement1 : "ActorManualMovement";
      statActorManualMovement2 : "ActorManualMovement";
      sudtActor1 : "typeActor";
      sudtActor2 : "typeActor";
      statManualWorkPos : Bool;
   END_VAR
BEGIN

REGION Network 1: Kamera einschalten / Switch on camera
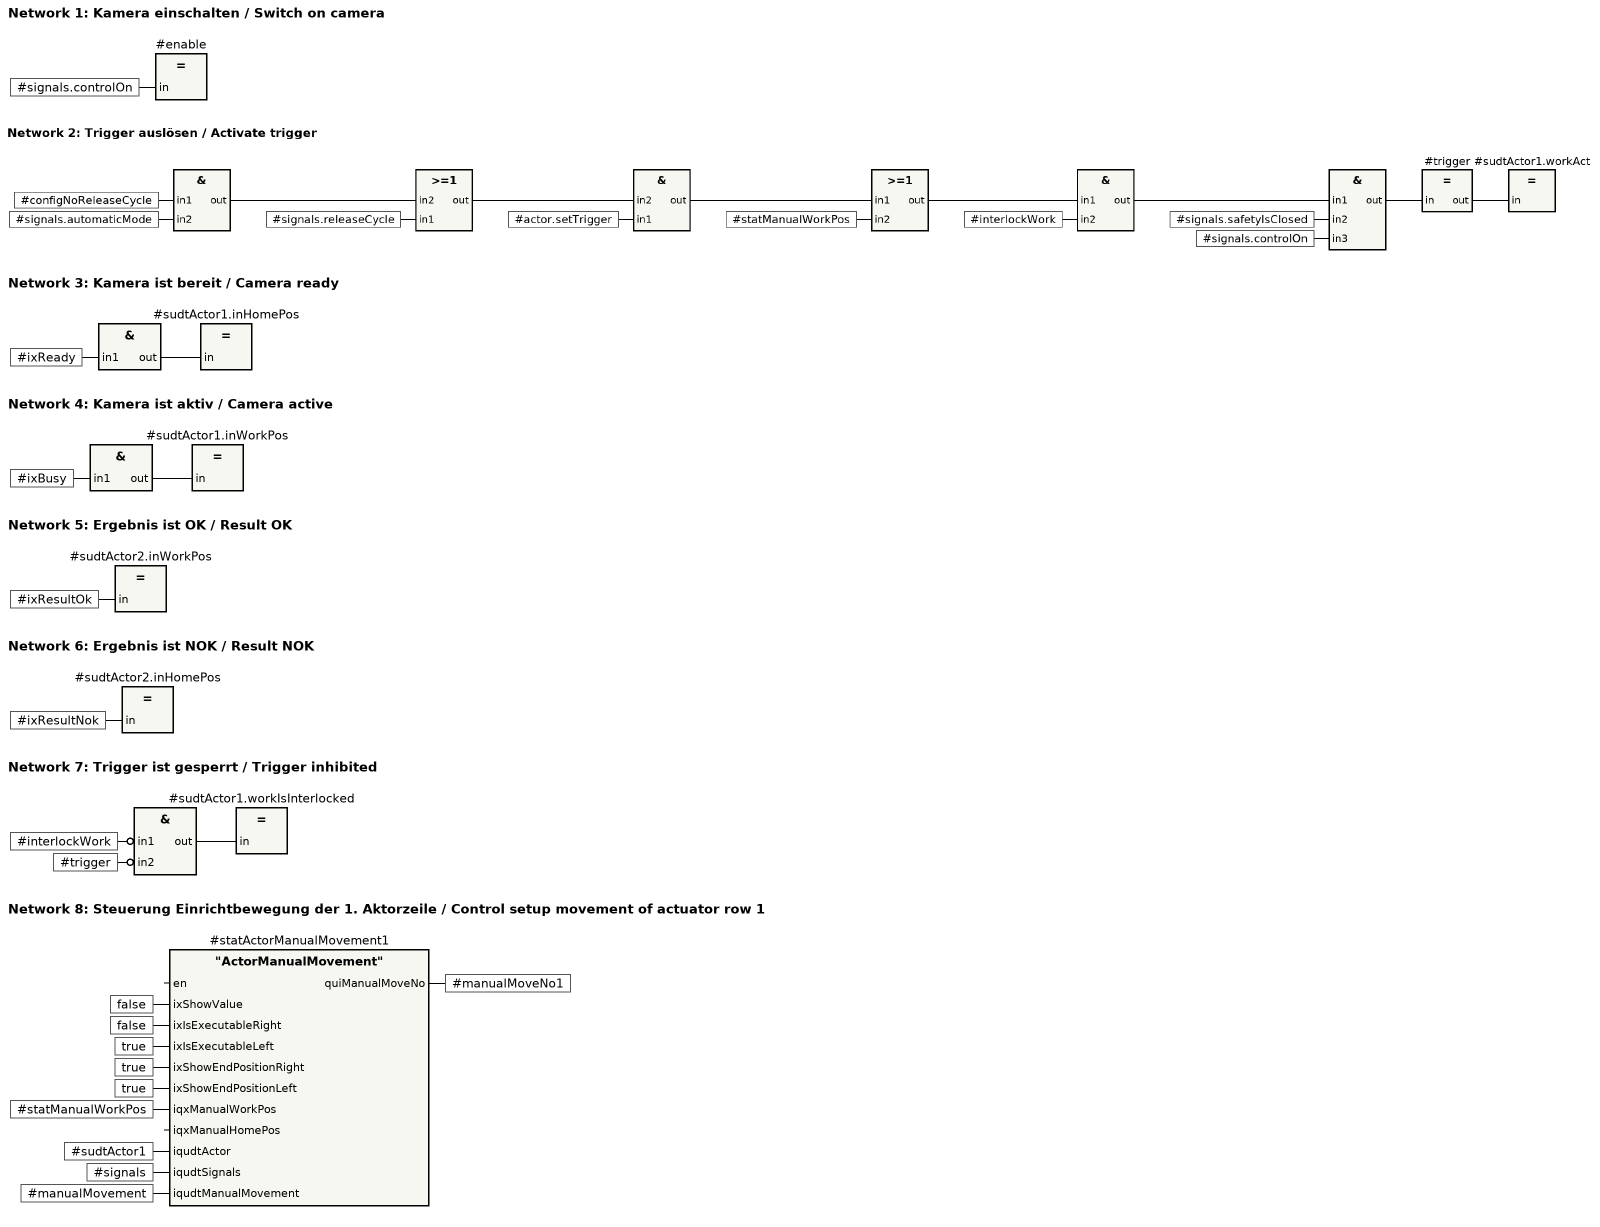
   #enable := #signals.controlOn;
END_REGION

REGION Network 2: Trigger auslösen / Activate trigger
   #trigger := ((((#configNoReleaseCycle AND #signals.automaticMode) OR #signals.releaseCycle) AND #actor.setTrigger) OR #statManualWorkPos) AND #interlockWork AND #signals.safetyIsClosed AND #signals.controlOn;
   #sudtActor1.workAct := #trigger;
END_REGION

REGION Network 3: Kamera ist bereit / Camera ready
   #sudtActor1.inHomePos := #ixReady;
END_REGION

REGION Network 4: Kamera ist aktiv / Camera active
   #sudtActor1.inWorkPos := #ixBusy;
END_REGION

REGION Network 5: Ergebnis ist OK / Result OK
   #sudtActor2.inWorkPos := #ixResultOk;
END_REGION

REGION Network 6: Ergebnis ist NOK / Result NOK
   #sudtActor2.inHomePos := #ixResultNok;
END_REGION

REGION Network 7: Trigger ist gesperrt / Trigger inhibited
   #sudtActor1.workIsInterlocked := NOT #interlockWork AND NOT #trigger;
END_REGION

REGION Network 8: Steuerung Einrichtbewegung der 1. Aktorzeile / Control setup movement of actuator row 1
   #statActorManualMovement1(ixShowValue := false,   // "ActorManualMovement"
                           ixIsExecutableRight := false,
                           ixIsExecutableLeft := true,
                           ixShowEndPositionRight := true,
                           ixShowEndPositionLeft := true,
                           iqxManualWorkPos := #statManualWorkPos,
                           iqudtActor := #sudtActor1,
                           iqudtSignals := #signals,
                           iqudtManualMovement := #manualMovement,
                           quiManualMoveNo => #manualMoveNo1);
END_REGION

REGION Network 9: Steuerung Einrichtbewegung der 2. Aktorzeile / Control setup movement of actuator row 2
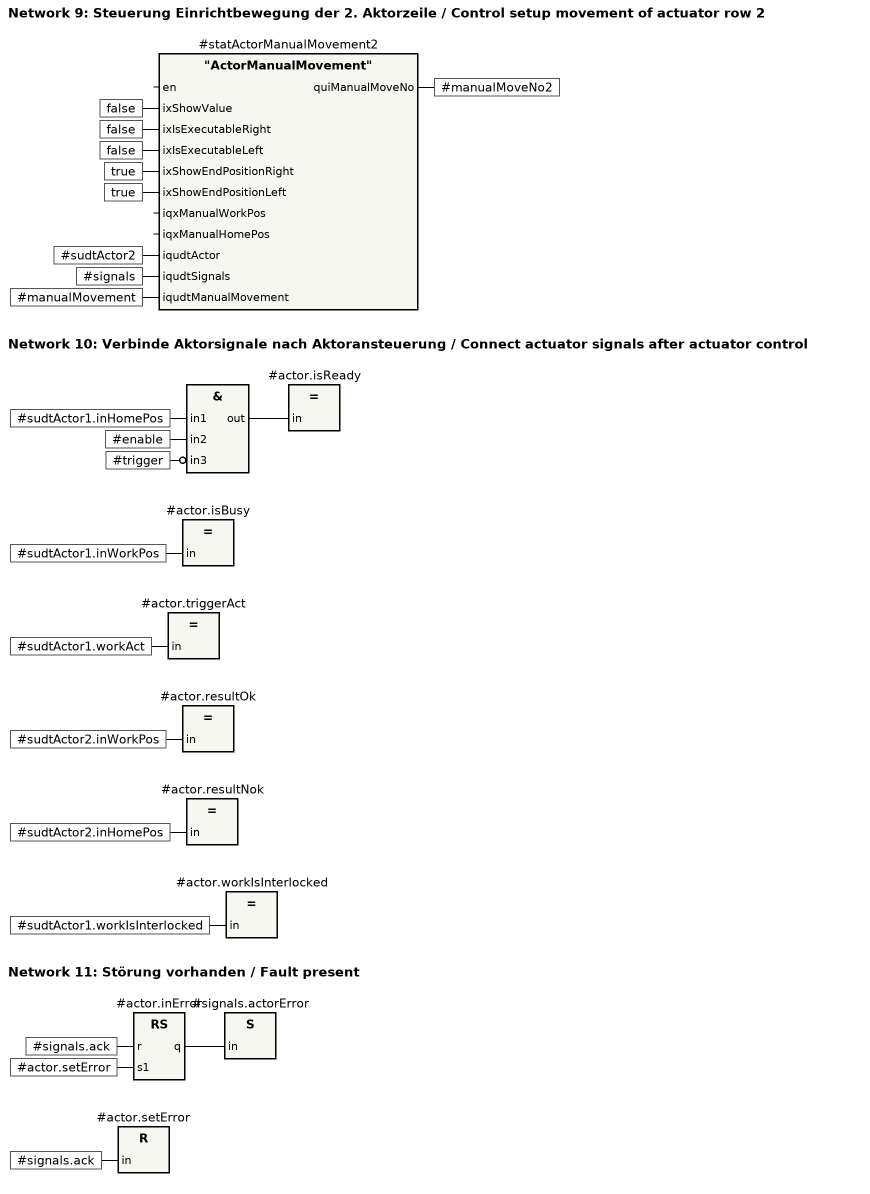
   #statActorManualMovement2(ixShowValue := false,   // "ActorManualMovement"
                           ixIsExecutableRight := false,
                           ixIsExecutableLeft := false,
                           ixShowEndPositionRight := true,
                           ixShowEndPositionLeft := true,
                           iqudtActor := #sudtActor2,
                           iqudtSignals := #signals,
                           iqudtManualMovement := #manualMovement,
                           quiManualMoveNo => #manualMoveNo2);
END_REGION

REGION Network 10: Verbinde Aktorsignale nach Aktoransteuerung / Connect actuator signals after actuator control
   #actor.isReady := #sudtActor1.inHomePos AND #enable AND NOT #trigger;
   #actor.isBusy := #sudtActor1.inWorkPos;
   #actor.triggerAct := #sudtActor1.workAct;
   #actor.resultOk := #sudtActor2.inWorkPos;
   #actor.resultNok := #sudtActor2.inHomePos;
   #actor.workIsInterlocked := #sudtActor1.workIsInterlocked;
END_REGION

REGION Network 11: Störung vorhanden / Fault present
   IF #signals.ack THEN
       #actor.inError := FALSE;   // RS flip-flop
   END_IF;
   IF #actor.setError THEN #actor.inError := TRUE; END_IF;
   IF #actor.inError THEN #signals.actorError := TRUE; END_IF;
   IF #signals.ack THEN #actor.setError := FALSE; END_IF;
END_REGION
END_FUNCTION_BLOCK

// folder: 9. Library/9.3 Processes

FUNCTION_BLOCK "Sq_Process_Stopper"   // FB9302, GRAPH_PLUS
{ S7_Optimized_Access := 'TRUE' }
VERSION : 0.1
   VAR_INPUT
      OFF_SQ : Bool := false;   // Kette ausschalten
      INIT_SQ : Bool := false;   // Kette in Initialzustand versetzen
      ACK_EF : Bool := false;   // Alle Fehler und Störungen quittieren
      S_PREV : Bool := false;   // Vorherigen Schritt am Parameter S_NO ausgeben
      S_NEXT : Bool := false;   // Nächsten Schritt am Parameter S_NO anzeigen
      SW_AUTO : Bool := false;   // Automatischer Betrieb
      SW_TAP : Bool := false;   // Halbautomatisch/Weiterschalten mit Transition
      SW_TOP : Bool := false;   // Halbautomatisch/Ignoriere Transition
      SW_MAN : Bool := false;   // Handbetrieb
      S_SEL : Int := 0;   // Schritt auswählen, der an S_NO ausgegeben werden soll
      S_ON : Bool := false;   // Schritt aktivieren, der an Parameter S_NO anliegt
      S_OFF : Bool := false;   // Schritt deaktivieren, der an Parameter S_NO anliegt
      T_PUSH : Bool := false;   // Schaltfreigabe für Transition im halbautomatischen Betrieb
      ixStart : Bool;   // Startfreigabe / Start enable
      ixCarrierPresent : Bool;   // WT am Stopper vorhanden / Workpiece carrier at stopper
      ixCheckTargetReached : Bool := false;   // 0 = Keine Sensor-Zielüberwachung nach Lift vorhanden / 0 = No destination sensor monitoring after lift
      ixTargetReached : Bool := false;   // WT-Sensor des nächsten Ziels / Workpiece carrier sensor at next destination
      itStopperRelease : Time := T#50ms;   // Zusätzliche Verzögerungszeit für Stopper öffnen, nachdem WT den Stopper verlassen hat / Additional stopper opening delay after workpiece carrier has left stopper
      itMaxRuntime : Time := t#5s;   // Maximale Laufzeit für diesen Prozess / Maximum execution time for this process
   END_VAR
   VAR_OUTPUT
      S_NO : Int := 0;   // Schrittnummer
      S_MORE : Bool := false;   // Weitere Schritte sind vorhanden und können in S_NO angezeigt werden.
      S_ACTIVE : Bool := false;   // Schritt, der an Parameter S_NO angezeigt wird, ist aktiv
      ERR_FLT : Bool := false;   // Sammelfehler Interlock oder Supervision
      AUTO_ON : Bool := false;   // Automatischer Betrieb eingeschaltet
      TAP_ON : Bool := false;   // Halbautomatischer Betrieb/Schritt mit Transition eingeschaltet
      TOP_ON : Bool := false;   // Halbautomatischer Betrieb/Ignoriere Transition eingeschaltet
      MAN_ON : Bool := false;   // Handbetrieb eingeschaltet
      qxWaitForTarget : Bool;   // Warte bis Ziel erreicht / Wait until destination reached
      qxIsActive : Bool;   // Prozess läuft / Process running
      qxIsInHome : Bool;   // steht in Grundstellung / in home position
   END_VAR
   VAR_IN_OUT
      signals : "typeStationSignals";   // Stationssteuersignale / Station control signals
      sq : "typeStepSequence";   // Schrittkettensteuersignale / Sequence control signals
      cylinder_stopper : "typeActor_1Out1In";   // Aktor für den Stopper / Stopper actuator
   END_VAR
   VAR
      sstReleaseCycle : Struct
         ErrorAck : Bool;
         No_LastCycle : Int;
         T : Time;   // Aktive Zeit des ReleaseCycle / Active time of ReleaseCycle
         Tck : Time;
         TckPrev : Time;
      END_STRUCT;
      HMI_INFO : Array[0..8] of UInt;
      IF_PAR : G7_IfParPlus_V6;
      RT_DATA : G7_RTDataPlus_V6;   // Interner Datenbereich
      Automatikablauf : G7_TransitionPlus_V6;   // Transitionsstruktur
      Freigabe : G7_TransitionPlus_V6;   // Transitionsstruktur
      Trans3 : G7_TransitionPlus_V6;   // Transitionsstruktur
      Fertig : G7_TransitionPlus_V6;   // Transitionsstruktur
      Grundstellungsfahrt : G7_TransitionPlus_V6;   // Transitionsstruktur
      GST_Aktiv : G7_TransitionPlus_V6;   // Transitionsstruktur
      GST_Beendet : G7_TransitionPlus_V6;   // Transitionsstruktur
      Beendet : G7_TransitionPlus_V6;   // Transitionsstruktur
      "WT hat Stopper verlassen" : G7_TransitionPlus_V6;   // Transitionsstruktur / Transition structure
      "Nachlaufzeit abgelaufen" : G7_TransitionPlus_V6;   // Transitionsstruktur / Transition structure
      "Ziel erreicht" : G7_TransitionPlus_V6;   // Transitionsstruktur / Transition structure
      Initialschritt : G7_StepPlus_V6;   // Schrittstruktur
      Grundstellung : G7_StepPlus_V6;   // Schrittstruktur
      SK_läuft : G7_StepPlus_V6;   // Schrittstruktur
      Fertigmeldung : G7_StepPlus_V6;   // Schrittstruktur
      "Start Grundstellungsfahrt" : G7_StepPlus_V6;   // Schrittstruktur
      "Fertig Grundstellungsfahrt" : G7_StepPlus_V6;   // Schrittstruktur
      Ende : G7_StepPlus_V6;   // Schrittstruktur
      "Stopper öffnen" : G7_StepPlus_V6;   // Schrittstruktur / Step structure
      Nachlaufzeit : G7_StepPlus_V6;   // Schrittstruktur / Step structure
      WaitForTarget : G7_StepPlus_V6;   // Schrittstruktur / Step structure
      SINI : Array[0..1] of USInt;
      LSTT : Array[0..10] of USInt;
      ATAJ : Array[0..10] of USInt;
      ATAB : Array[0..10] of USInt;
      PSTT : Array[0..10] of USInt;
      NSTT : Array[0..10] of USInt;
      ASSJ : Array[0..9] of USInt;
      ASSB : Array[0..9] of USInt;
      PTTS : Array[0..9] of USInt;
      NTTS : Array[0..9] of USInt;
      SW_SQTS : Array[0..9] of USInt;
      SWITCH : Array[0..1] of USInt;
      TVX : Array[0..3] of USInt;
      TTX : Array[0..3] of USInt;
      TSX : Array[0..1] of USInt;
      S00X : Array[0..1] of USInt;
      SOFFX : Array[0..1] of USInt;
      SONX : Array[0..1] of USInt;
      SAX : Array[0..1] of USInt;
      SERRX : Array[0..10] of USInt;
      SMX : Array[0..10] of USInt;
      S0X : Array[0..10] of USInt;
      S1X : Array[0..10] of USInt;
      IL_ALARM_INST : Diag_Alarm;
      SUP_ALARM_INST : Diag_Alarm;
      STEP_TIME_ALARM_INST : Diag_Alarm;
      IEC_TIMER_INST : IEC_TIMER;
      TRANSACTION_FLAG : Bool := false;
   END_VAR
   VAR_TEMP
      txStartCondition : Bool;
      tdTckDiff : DInt;
   END_VAR
   VAR_TEMP   // added for the SCL form of the ladder/FBD networks
      _w1 : Bool;
      _w2 : Bool;
   END_VAR
   // SINI[0] := 2;
   // LSTT[0] := 255;
   // LSTT[1] := 255;
   // LSTT[2] := 255;
   // LSTT[3] := 255;
   // LSTT[4] := 255;
   // LSTT[5] := 255;
   // LSTT[6] := 255;
   // LSTT[7] := 1;
   // ATAJ[1] := 1;
   // ATAJ[2] := 2;
   // ATAJ[3] := 6;
   // ATAJ[4] := 4;
   // ATAJ[5] := 5;
   // ATAJ[6] := 3;
   // ATAJ[7] := 7;
   // ATAB[0] := 4;
   // ATAB[1] := 1;
   // ATAB[2] := 2;
   // ATAB[3] := 3;
   // ATAB[5] := 5;
   // ATAB[6] := 6;
   // ATAB[7] := 7;
   // PSTT[1] := 1;
   // PSTT[2] := 2;
   // PSTT[3] := 3;
   // PSTT[5] := 4;
   // PSTT[6] := 5;
   // PSTT[7] := 6;
   // NSTT[0] := 1;
   // NSTT[1] := 2;
   // NSTT[2] := 7;
   // NSTT[3] := 6;
   // NSTT[4] := 4;
   // NSTT[5] := 5;
   // NSTT[6] := 6;
   // NSTT[7] := 1;
   // ASSJ[1] := 1;
   // ASSJ[2] := 2;
   // ASSJ[3] := 3;
   // ASSJ[4] := 4;
   // ASSJ[5] := 5;
   // ASSJ[6] := 6;
   // ASSB[1] := 1;
   // ASSB[2] := 2;
   // ASSB[3] := 3;
   // ASSB[4] := 4;
   // ASSB[5] := 5;
   // ASSB[6] := 6;
   // PTTS[0] := 255;
   // PTTS[2] := 1;
   // PTTS[3] := 10;
   // PTTS[4] := 4;
   // PTTS[5] := 5;
   // PTTS[6] := 3;
   // NTTS[1] := 1;
   // NTTS[2] := 2;
   // NTTS[3] := 3;
   // NTTS[4] := 5;
   // NTTS[5] := 6;
   // NTTS[6] := 7;
   // SW_SQTS[1] := 1;
   // SW_SQTS[2] := 1;
   // SW_SQTS[3] := 1;
   // SW_SQTS[4] := 2;
   // SW_SQTS[5] := 2;
   // SW_SQTS[6] := 3;
   // TVX[0] := 16#1;
   // TTX[0] := 16#1;
   // TSX[0] := 16#1;
   // S00X[0] := 16#1;
   // SOFFX[0] := 16#1;
   // SONX[0] := 16#1;
   // SAX[0] := 16#1;
   // SERRX[0] := 16#1;
   // SMX[0] := 16#1;
   // S0X[0] := 16#1;
   // S1X[0] := 16#1;
   // LSTT[8] := 255;
   // ATAJ[8] := 8;
   // ATAB[8] := 8;
   // PSTT[8] := 7;
   // NSTT[8] := 8;
   // ASSJ[7] := 7;
   // ASSB[7] := 7;
   // PTTS[7] := 2;
   // NTTS[7] := 8;
   // SW_SQTS[7] := 1;
   // LSTT[9] := 255;
   // LSTT[10] := 255;
   // ATAJ[9] := 9;
   // ATAJ[10] := 10;
   // ATAB[9] := 9;
   // ATAB[10] := 10;
   // PSTT[9] := 8;
   // PSTT[10] := 9;
   // NSTT[9] := 9;
   // NSTT[10] := 3;
   // ASSJ[8] := 8;
   // ASSJ[9] := 9;
   // ASSB[8] := 8;
   // ASSB[9] := 9;
   // PTTS[8] := 8;
   // PTTS[9] := 9;
   // NTTS[8] := 9;
   // NTTS[9] := 10;
   // SW_SQTS[8] := 1;
   // SW_SQTS[9] := 1;
BEGIN
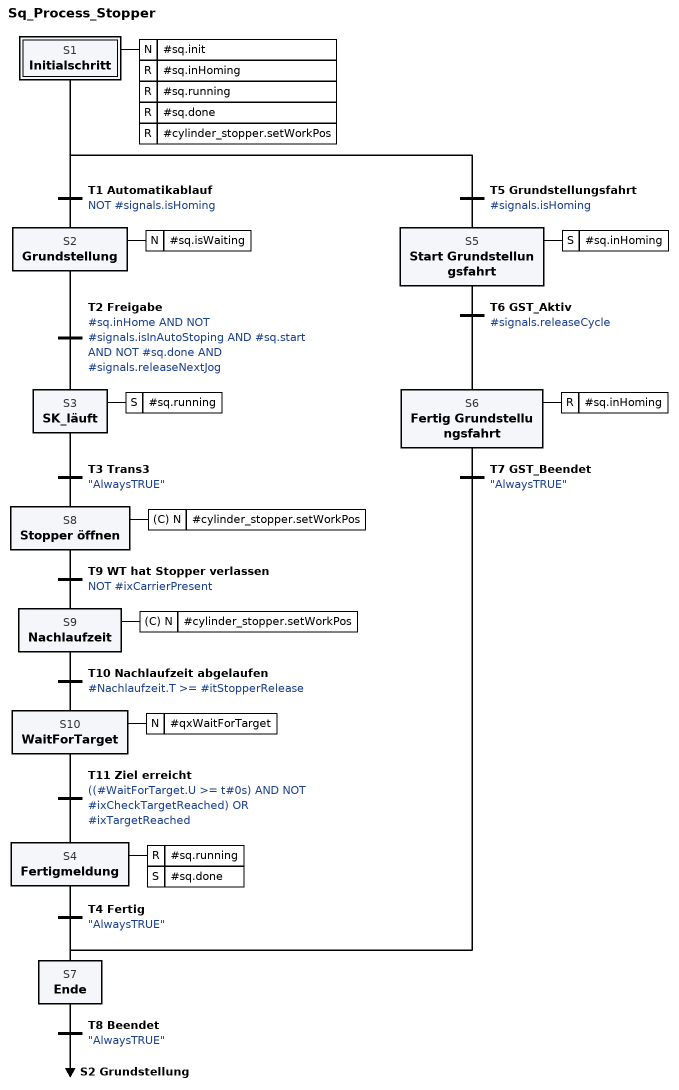
   // permanent pre-instructions
   NETWORK 1
   TITLE = Schrittkette verfügbar / Sequence available
      #sq.exists := true;
   NETWORK 2
   TITLE = Schrittkette in Grundstellung (Erweitern) / Sequence in home position (extend)
      #sq.inHome := #Grundstellung.X AND #cylinder_stopper.inHomePos;
   NETWORK 3
   TITLE = Startbedingung (Erweitern) / Start condition (extend)
      #txStartCondition := (NOT #ixCheckTargetReached OR NOT #ixTargetReached) AND #ixStart AND #ixCarrierPresent;
   NETWORK 4
   TITLE = Schrittkette starten / Start sequence
      #sq.start := #sq.inHome AND NOT #sq.running AND #signals.releaseCycle AND NOT #signals.isHoming AND #txStartCondition;
      IF #sq.start THEN #sq.done := FALSE; END_IF;
   NETWORK 5
   TITLE = ReleaseCycle-Zeitgeber / ReleaseCycle timer
      // ENO of a box is taken as its EN; it also drops when the box reports an error
      #_w1 := #ERR_FLT AND #ACK_EF;
      #_w2 := #_w1 AND NOT #sstReleaseCycle.ErrorAck;   // rising edge
      #sstReleaseCycle.ErrorAck := #_w1;
      IF (#S_NO <> #sstReleaseCycle.No_LastCycle) OR #_w2 THEN
          #sstReleaseCycle.T := T#0MS;
          #sstReleaseCycle.TckPrev := #sstReleaseCycle.Tck;
          #sstReleaseCycle.No_LastCycle := #S_NO;
      END_IF;
      #sstReleaseCycle.Tck := TIME_TCK();
      #tdTckDiff := #sstReleaseCycle.Tck - #sstReleaseCycle.TckPrev;
      #sstReleaseCycle.TckPrev := #sstReleaseCycle.Tck;
      IF (0 <= #tdTckDiff) AND (#tdTckDiff <= 1000) AND #signals.releaseCycle THEN
          #sstReleaseCycle.T := #sstReleaseCycle.T + #tdTckDiff;
      END_IF;

   // sequencer 1
   INITIAL_STEP Initialschritt:   // S1, max time T#10S, warning time T#7S
              N    #sq.init
              R    #sq.inHoming
              R    #sq.running
              R    #sq.done
              R    #cylinder_stopper.setWorkPos
   END_STEP
   TRANSITION Automatikablauf FROM Initialschritt TO Grundstellung   // T1
      := NOT #signals.isHoming;
   END_TRANSITION
   TRANSITION Grundstellungsfahrt FROM Initialschritt TO "Start Grundstellungsfahrt"   // T5
      := #signals.isHoming;
   END_TRANSITION
   STEP Grundstellung:   // S2, max time T#10S, warning time T#7S
              N    #sq.isWaiting
   END_STEP
   TRANSITION Freigabe FROM Grundstellung TO SK_läuft   // T2
      := #sq.inHome AND NOT #signals.isInAutoStoping AND #sq.start AND NOT #sq.done AND #signals.releaseNextJog;
   END_TRANSITION
   STEP SK_läuft:   // S3, max time T#10S, warning time T#7S
              S    #sq.running
   END_STEP
   TRANSITION Trans3 FROM SK_läuft TO "Stopper öffnen"   // T3
      := "AlwaysTRUE";
   END_TRANSITION
   STEP Fertigmeldung:   // S4, max time T#10S, warning time T#7S
              R    #sq.running
              S    #sq.done
   END_STEP
   TRANSITION Fertig FROM Fertigmeldung TO Ende   // T4
      := "AlwaysTRUE";
   END_TRANSITION
   STEP "Start Grundstellungsfahrt":   // S5, max time T#10S, warning time T#7S
              S    #sq.inHoming
   END_STEP
   TRANSITION GST_Aktiv FROM "Start Grundstellungsfahrt" TO "Fertig Grundstellungsfahrt"   // T6
      := #signals.releaseCycle;
   END_TRANSITION
   STEP "Fertig Grundstellungsfahrt":   // S6, max time T#10S, warning time T#7S
              R    #sq.inHoming
   END_STEP
   TRANSITION GST_Beendet FROM "Fertig Grundstellungsfahrt" TO Ende   // T7
      := "AlwaysTRUE";
   END_TRANSITION
   STEP Ende:   // S7, max time T#10S, warning time T#7S
   END_STEP
   TRANSITION Beendet FROM Ende TO Grundstellung   // T8, jump
      := "AlwaysTRUE";
   END_TRANSITION
   STEP "Stopper öffnen":   // S8, max time T#10S, warning time T#7S
      supervision V := #sstReleaseCycle.T >= #itMaxRuntime;
      (C)     N    #cylinder_stopper.setWorkPos
   END_STEP
   TRANSITION "WT hat Stopper verlassen" FROM "Stopper öffnen" TO Nachlaufzeit   // T9
      := NOT #ixCarrierPresent;
   END_TRANSITION
   STEP Nachlaufzeit:   // S9, max time T#10S, warning time T#7S
      (C)     N    #cylinder_stopper.setWorkPos
   END_STEP
   TRANSITION "Nachlaufzeit abgelaufen" FROM Nachlaufzeit TO WaitForTarget   // T10
      := #Nachlaufzeit.T >= #itStopperRelease;
   END_TRANSITION
   STEP WaitForTarget:   // S10, max time T#10S, warning time T#7S
      supervision V := #sstReleaseCycle.T >= #itMaxRuntime;
              N    #qxWaitForTarget
   END_STEP
   TRANSITION "Ziel erreicht" FROM WaitForTarget TO Fertigmeldung   // T11
      := ((#WaitForTarget.U >= t#0s) AND NOT #ixCheckTargetReached) OR #ixTargetReached;
   END_TRANSITION

   // permanent post-instructions
   NETWORK 1
   TITLE = Störungssignal weitergeben / Forward fault signal
      #sq.error := #ERR_FLT;
   NETWORK 2
   TITLE = Ablauf ist aktiv / Sequence active
      #qxIsActive := #sq.running;
   NETWORK 3
   TITLE = steht in Grundstellung / in home position
      #qxIsInHome := #sq.inHome AND NOT #sq.running;
END_FUNCTION_BLOCK

FUNCTION_BLOCK "Sq_Process_Lift"   // FB9303, GRAPH_PLUS
{ S7_Optimized_Access := 'TRUE' }
VERSION : 0.1
   VAR_INPUT
      OFF_SQ : Bool := false;   // Kette ausschalten
      INIT_SQ : Bool := false;   // Kette in Initialzustand versetzen
      ACK_EF : Bool := false;   // Alle Fehler und Störungen quittieren
      S_PREV : Bool := false;   // Vorherigen Schritt am Parameter S_NO ausgeben
      S_NEXT : Bool := false;   // Nächsten Schritt am Parameter S_NO anzeigen
      SW_AUTO : Bool := false;   // Automatischer Betrieb
      SW_TAP : Bool := false;   // Halbautomatisch/Weiterschalten mit Transition
      SW_TOP : Bool := false;   // Halbautomatisch/Ignoriere Transition
      SW_MAN : Bool := false;   // Handbetrieb
      S_SEL : Int := 0;   // Schritt auswählen, der an S_NO ausgegeben werden soll
      S_ON : Bool := false;   // Schritt aktivieren, der an Parameter S_NO anliegt
      S_OFF : Bool := false;   // Schritt deaktivieren, der an Parameter S_NO anliegt
      T_PUSH : Bool := false;   // Schaltfreigabe für Transition im halbautomatischen Betrieb
      ixExternReqConvIn : Bool;   // Externe Anforderung Förderband Einlauf starten / External request to start infeed conveyor
      ixCarrierPresent : Bool;   // WT auf dem Lift vorhanden / Workpiece carrier present on lift
      ixCheckTargetReached : Bool := false;   // 0 = Keine Sensor-Zielüberwachung nach Lift vorhanden / 0 = No destination sensor monitoring after lift
      ixTargetReached : Bool := false;   // WT-Sensor des nächsten Ziels / Workpiece carrier sensor at next destination
      itCarrierReactionDelay : Time := T#350ms;   // Verzögerungszeit für die WT-Erkennung / Workpiece carrier detection delay
      itMaxRuntime : Time := t#10s;   // Maximale Laufzeit für diesen Prozess / Maximum execution time for this process
   END_VAR
   VAR_OUTPUT
      S_NO : Int := 0;   // Schrittnummer
      S_MORE : Bool := false;   // Weitere Schritte sind vorhanden und können in S_NO angezeigt werden.
      S_ACTIVE : Bool := false;   // Schritt, der an Parameter S_NO angezeigt wird, ist aktiv
      ERR_FLT : Bool := false;   // Sammelfehler Interlock oder Supervision
      AUTO_ON : Bool := false;   // Automatischer Betrieb eingeschaltet
      TAP_ON : Bool := false;   // Halbautomatischer Betrieb/Schritt mit Transition eingeschaltet
      TOP_ON : Bool := false;   // Halbautomatischer Betrieb/Ignoriere Transition eingeschaltet
      MAN_ON : Bool := false;   // Handbetrieb eingeschaltet
      qxIsActive : Bool;   // Schrittkette läuft / Sequence running
      qxIsInHome : Bool;   // steht in Grundstellung / in home position
      qxReadyForNextWT : Bool;   // Bereit für den nächsten WT / Ready for next workpiece carrier
      qxTransfered : Bool;   // WT wurde abtransportiert (1-Zyklus true) / Workpiece carrier transported away (true for one cycle)
   END_VAR
   VAR_IN_OUT
      signals : "typeStationSignals";   // Stationssteuersignale / Station control signals
      sq : "typeStepSequence";   // Schrittkettensteuersignale / Sequence control signals
      cylinder : "typeActor_2Out2In";   // Aktor des Zylinders für den Lift / Lift cylinder actuator
      conveyor : "typeActor_2Out0In";   // Aktor des Förderbands für den Lift / Lift conveyor actuator
   END_VAR
   VAR
      sstReleaseCycle : Struct
         ErrorAck : Bool;
         No_LastCycle : Int;
         T : Time;   // Aktive Zeit des ReleaseCycle / Active time of ReleaseCycle
         Tck : Time;
         TckPrev : Time;
      END_STRUCT;
      sinstCarrierOnLift : TON_TIME;
      sinstCarrierLeftLift : TON_TIME;
      susiLiftState : USInt;
      HMI_INFO : Array[0..8] of UInt;
      IF_PAR : G7_IfParPlus_V6;
      RT_DATA : G7_RTDataPlus_V6;   // Interner Datenbereich
      Automatikablauf : G7_TransitionPlus_V6;   // Transitionsstruktur
      Freigabe : G7_TransitionPlus_V6;   // Transitionsstruktur
      Trans3 : G7_TransitionPlus_V6;   // Transitionsstruktur
      Fertig : G7_TransitionPlus_V6;   // Transitionsstruktur
      Grundstellungsfahrt : G7_TransitionPlus_V6;   // Transitionsstruktur
      GST_Aktiv : G7_TransitionPlus_V6;   // Transitionsstruktur
      GST_Beendet : G7_TransitionPlus_V6;   // Transitionsstruktur
      Beendet : G7_TransitionPlus_V6;   // Transitionsstruktur
      "WT ist komplett auf dem Lift eingefahren" : G7_TransitionPlus_V6;   // Transitionsstruktur / Transition structure
      "WT ist komplett auf dem Lift eingefahren_1" : G7_TransitionPlus_V6;   // Transitionsstruktur / Transition structure
      "Wt hat den Lift verlassen" : G7_TransitionPlus_V6;   // Transitionsstruktur / Transition structure
      "Lift steht in Arbeitsstellung" : G7_TransitionPlus_V6;   // Transitionsstruktur / Transition structure
      "Wt hat Endziel erreicht" : G7_TransitionPlus_V6;   // Transitionsstruktur / Transition structure
      "Lift steht in Grundstellung" : G7_TransitionPlus_V6;   // Transitionsstruktur / Transition structure
      GS_LiftInHome : G7_TransitionPlus_V6;   // Transitionsstruktur / Transition structure
      GS_LiftInWork : G7_TransitionPlus_V6;   // Transitionsstruktur / Transition structure
      LiftIsEmpty : G7_TransitionPlus_V6;   // Transitionsstruktur / Transition structure
      "Endziel ist frei" : G7_TransitionPlus_V6;   // Transitionsstruktur / Transition structure
      "Endziel ist belegt" : G7_TransitionPlus_V6;   // Transitionsstruktur / Transition structure
      GS_NoWtOnLift : G7_TransitionPlus_V6;   // Transitionsstruktur / Transition structure
      GS_WtOnLift : G7_TransitionPlus_V6;   // Transitionsstruktur / Transition structure
      GS_LiftEmpty : G7_TransitionPlus_V6;   // Transitionsstruktur / Transition structure
      GS_LiftBusy : G7_TransitionPlus_V6;   // Transitionsstruktur / Transition structure
      LiftIsBusy : G7_TransitionPlus_V6;   // Transitionsstruktur / Transition structure
      State_LiftBusy : G7_TransitionPlus_V6;   // Transitionsstruktur / Transition structure
      State_LiftEmpty : G7_TransitionPlus_V6;   // Transitionsstruktur / Transition structure
      JogT1 : G7_TransitionPlus_V6;   // Transitionsstruktur / Transition structure
      JogT2 : G7_TransitionPlus_V6;   // Transitionsstruktur / Transition structure
      JogT3 : G7_TransitionPlus_V6;   // Transitionsstruktur / Transition structure
      Initialschritt : G7_StepPlus_V6;   // Schrittstruktur
      Grundstellung : G7_StepPlus_V6;   // Schrittstruktur
      SK_läuft : G7_StepPlus_V6;   // Schrittstruktur
      Fertigmeldung : G7_StepPlus_V6;   // Schrittstruktur
      "Start Grundstellungsfahrt" : G7_StepPlus_V6;   // Schrittstruktur
      "Fertig Grundstellungsfahrt" : G7_StepPlus_V6;   // Schrittstruktur
      Ende : G7_StepPlus_V6;   // Schrittstruktur
      ConvIn : G7_StepPlus_V6;   // Schrittstruktur / Step structure
      GS_ConvIn : G7_StepPlus_V6;   // Schrittstruktur / Step structure
      ConvOut : G7_StepPlus_V6;   // Schrittstruktur / Step structure
      LiftToWork : G7_StepPlus_V6;   // Schrittstruktur / Step structure
      WaitConvOut : G7_StepPlus_V6;   // Schrittstruktur / Step structure
      LiftToHome : G7_StepPlus_V6;   // Schrittstruktur / Step structure
      GS_CylHome : G7_StepPlus_V6;   // Schrittstruktur / Step structure
      GS_CylWork : G7_StepPlus_V6;   // Schrittstruktur / Step structure
      Warte_Endziel_frei : G7_StepPlus_V6;   // Schrittstruktur / Step structure
      GS_CheckSensor : G7_StepPlus_V6;   // Schrittstruktur / Step structure
      GS_StateEmpty : G7_StepPlus_V6;   // Schrittstruktur / Step structure
      GS_StateBusy : G7_StepPlus_V6;   // Schrittstruktur / Step structure
      CheckState : G7_StepPlus_V6;   // Schrittstruktur / Step structure
      StateBusy : G7_StepPlus_V6;   // Schrittstruktur / Step structure
      StateEmpty : G7_StepPlus_V6;   // Schrittstruktur / Step structure
      JogS1 : G7_StepPlus_V6;   // Schrittstruktur / Step structure
      JogS2 : G7_StepPlus_V6;   // Schrittstruktur / Step structure
      JogS3 : G7_StepPlus_V6;   // Schrittstruktur / Step structure
      SINI : Array[0..1] of USInt;
      LSTT : Array[0..28] of USInt;
      ATAJ : Array[0..28] of USInt;
      ATAB : Array[0..28] of USInt;
      PSTT : Array[0..28] of USInt;
      NSTT : Array[0..28] of USInt;
      ASSJ : Array[0..24] of USInt;
      ASSB : Array[0..24] of USInt;
      PTTS : Array[0..24] of USInt;
      NTTS : Array[0..24] of USInt;
      SW_SQTS : Array[0..24] of USInt;
      SWITCH : Array[0..15] of USInt;
      TVX : Array[0..9] of USInt;
      TTX : Array[0..9] of USInt;
      TSX : Array[0..1] of USInt;
      S00X : Array[0..1] of USInt;
      SOFFX : Array[0..1] of USInt;
      SONX : Array[0..1] of USInt;
      SAX : Array[0..1] of USInt;
      SERRX : Array[0..25] of USInt;
      SMX : Array[0..25] of USInt;
      S0X : Array[0..25] of USInt;
      S1X : Array[0..25] of USInt;
      IL_ALARM_INST : Diag_Alarm;
      SUP_ALARM_INST : Diag_Alarm;
      STEP_TIME_ALARM_INST : Diag_Alarm;
      IEC_TIMER_INST : IEC_TIMER;
      TRANSACTION_FLAG : Bool := false;
   END_VAR
   VAR_TEMP
      txStartCondition : Bool;
      tdTckDiff : DInt;
   END_VAR
   VAR CONSTANT
      LIFT_UNKOWN : USInt := 0;   // Zustand unbekannt / State unknown
      LIFT_EMPTY : USInt := 1;   // Kein WT auf dem Lift / No workpiece carrier on lift
      LIFT_BUSY : USInt := 2;   // WT auf Lift vorhanden / Workpiece carrier present on lift
   END_VAR
   VAR_TEMP   // added for the SCL form of the ladder/FBD networks
      _w1 : Bool;
      _w2 : Bool;
   END_VAR
   // SINI[0] := 2;
   // LSTT[0] := 255;
   // LSTT[1] := 255;
   // LSTT[2] := 255;
   // LSTT[3] := 255;
   // LSTT[4] := 255;
   // LSTT[5] := 255;
   // LSTT[6] := 255;
   // LSTT[7] := 1;
   // ATAJ[1] := 1;
   // ATAJ[2] := 2;
   // ATAJ[3] := 6;
   // ATAJ[4] := 4;
   // ATAJ[5] := 5;
   // ATAJ[6] := 3;
   // ATAJ[7] := 7;
   // ATAB[0] := 4;
   // ATAB[1] := 1;
   // ATAB[2] := 2;
   // ATAB[3] := 3;
   // ATAB[5] := 5;
   // ATAB[6] := 6;
   // ATAB[7] := 7;
   // PSTT[1] := 1;
   // PSTT[2] := 2;
   // PSTT[3] := 3;
   // PSTT[5] := 4;
   // PSTT[6] := 5;
   // PSTT[7] := 6;
   // NSTT[0] := 1;
   // NSTT[1] := 2;
   // NSTT[2] := 19;
   // NSTT[3] := 6;
   // NSTT[4] := 4;
   // NSTT[5] := 8;
   // NSTT[6] := 6;
   // NSTT[7] := 1;
   // ASSJ[1] := 1;
   // ASSJ[2] := 2;
   // ASSJ[3] := 3;
   // ASSJ[4] := 4;
   // ASSJ[5] := 5;
   // ASSJ[6] := 6;
   // ASSB[1] := 1;
   // ASSB[2] := 2;
   // ASSB[3] := 3;
   // ASSB[4] := 4;
   // ASSB[5] := 5;
   // ASSB[6] := 6;
   // PTTS[0] := 255;
   // PTTS[2] := 1;
   // PTTS[3] := 13;
   // PTTS[4] := 4;
   // PTTS[5] := 14;
   // PTTS[6] := 3;
   // NTTS[1] := 1;
   // NTTS[2] := 2;
   // NTTS[3] := 3;
   // NTTS[4] := 5;
   // NTTS[5] := 6;
   // NTTS[6] := 7;
   // SW_SQTS[1] := 1;
   // SW_SQTS[2] := 1;
   // SW_SQTS[3] := 2;
   // SW_SQTS[4] := 3;
   // SW_SQTS[5] := 4;
   // SW_SQTS[6] := 5;
   // TVX[0] := 16#1;
   // TTX[0] := 16#1;
   // TSX[0] := 16#1;
   // S00X[0] := 16#1;
   // SOFFX[0] := 16#1;
   // SONX[0] := 16#1;
   // SAX[0] := 16#1;
   // SERRX[0] := 16#1;
   // SMX[0] := 16#1;
   // S0X[0] := 16#1;
   // S1X[0] := 16#1;
   // LSTT[8] := 255;
   // ATAJ[8] := 8;
   // ATAB[8] := 8;
   // PSTT[8] := 7;
   // NSTT[8] := 20;
   // ASSJ[7] := 7;
   // ASSB[7] := 7;
   // PTTS[7] := 16;
   // NTTS[7] := 8;
   // SW_SQTS[7] := 6;
   // LSTT[9] := 255;
   // LSTT[10] := 255;
   // LSTT[11] := 255;
   // ATAJ[9] := 9;
   // ATAJ[10] := 10;
   // ATAJ[11] := 11;
   // ATAB[9] := 9;
   // ATAB[10] := 10;
   // ATAB[11] := 11;
   // PSTT[9] := 8;
   // PSTT[10] := 9;
   // PSTT[11] := 10;
   // NSTT[9] := 16;
   // NSTT[10] := 11;
   // NSTT[11] := 23;
   // ASSJ[8] := 8;
   // ASSJ[9] := 9;
   // ASSJ[10] := 10;
   // ASSB[8] := 8;
   // ASSB[9] := 9;
   // ASSB[10] := 10;
   // PTTS[8] := 5;
   // PTTS[9] := 17;
   // PTTS[10] := 26;
   // NTTS[8] := 9;
   // NTTS[9] := 10;
   // NTTS[10] := 11;
   // SW_SQTS[8] := 3;
   // SW_SQTS[9] := 7;
   // SW_SQTS[10] := 8;
   // LSTT[12] := 255;
   // LSTT[13] := 255;
   // ATAJ[12] := 12;
   // ATAJ[13] := 18;
   // ATAB[12] := 12;
   // ATAB[13] := 13;
   // PSTT[12] := 11;
   // PSTT[13] := 12;
   // NSTT[12] := 21;
   // NSTT[13] := 3;
   // ASSJ[11] := 11;
   // ASSJ[12] := 12;
   // ASSB[11] := 11;
   // ASSB[12] := 12;
   // PTTS[11] := 10;
   // PTTS[12] := 28;
   // NTTS[11] := 12;
   // NTTS[12] := 13;
   // SW_SQTS[11] := 7;
   // SW_SQTS[12] := 7;
   // LSTT[14] := 255;
   // LSTT[15] := 255;
   // ATAJ[14] := 15;
   // ATAJ[15] := 14;
   // ATAB[14] := 14;
   // ATAB[15] := 15;
   // PSTT[14] := 13;
   // PSTT[15] := 14;
   // NSTT[14] := 5;
   // NSTT[15] := 5;
   // ASSJ[13] := 13;
   // ASSJ[14] := 14;
   // ASSB[13] := 13;
   // ASSB[14] := 14;
   // PTTS[13] := 21;
   // PTTS[14] := 22;
   // NTTS[13] := 14;
   // NTTS[14] := 15;
   // SW_SQTS[13] := 9;
   // SW_SQTS[14] := 10;
   // LSTT[16] := 255;
   // LSTT[17] := 255;
   // ATAJ[16] := 16;
   // ATAJ[17] := 17;
   // ATAB[16] := 23;
   // ATAB[17] := 18;
   // PSTT[16] := 19;
   // PSTT[17] := 15;
   // NSTT[16] := 7;
   // NSTT[17] := 9;
   // ASSJ[15] := 15;
   // ASSJ[16] := 16;
   // ASSB[15] := 15;
   // ASSB[16] := 16;
   // PTTS[15] := 27;
   // PTTS[16] := 9;
   // NTTS[15] := 17;
   // NTTS[16] := 19;
   // SW_SQTS[15] := 8;
   // SW_SQTS[16] := 3;
   // LSTT[18] := 255;
   // LSTT[19] := 255;
   // ATAJ[18] := 13;
   // ATAJ[19] := 19;
   // ATAB[18] := 17;
   // ATAB[19] := 20;
   // PSTT[18] := 15;
   // PSTT[19] := 16;
   // NSTT[18] := 3;
   // NSTT[19] := 17;
   // ASSJ[17] := 17;
   // ASSB[17] := 17;
   // PTTS[17] := 19;
   // NTTS[17] := 21;
   // SW_SQTS[17] := 9;
   // LSTT[20] := 255;
   // LSTT[21] := 255;
   // LSTT[22] := 255;
   // LSTT[23] := 255;
   // LSTT[24] := 255;
   // LSTT[25] := 255;
   // LSTT[26] := 255;
   // LSTT[27] := 255;
   // LSTT[28] := 255;
   // ATAJ[20] := 20;
   // ATAJ[21] := 21;
   // ATAJ[22] := 22;
   // ATAJ[23] := 26;
   // ATAJ[24] := 24;
   // ATAJ[25] := 25;
   // ATAJ[26] := 23;
   // ATAJ[27] := 27;
   // ATAJ[28] := 28;
   // ATAB[20] := 19;
   // ATAB[21] := 21;
   // ATAB[22] := 22;
   // ATAB[23] := 16;
   // ATAB[24] := 24;
   // ATAB[25] := 25;
   // ATAB[26] := 26;
   // ATAB[27] := 27;
   // ATAB[28] := 28;
   // PSTT[20] := 16;
   // PSTT[21] := 17;
   // PSTT[22] := 18;
   // PSTT[23] := 19;
   // PSTT[24] := 20;
   // PSTT[25] := 21;
   // PSTT[26] := 22;
   // PSTT[27] := 23;
   // PSTT[28] := 24;
   // NSTT[20] := 18;
   // NSTT[21] := 13;
   // NSTT[22] := 14;
   // NSTT[23] := 10;
   // NSTT[24] := 22;
   // NSTT[25] := 24;
   // NSTT[26] := 10;
   // NSTT[27] := 15;
   // NSTT[28] := 12;
   // ASSJ[18] := 18;
   // ASSJ[19] := 19;
   // ASSJ[20] := 20;
   // ASSJ[21] := 21;
   // ASSJ[22] := 22;
   // ASSJ[23] := 23;
   // ASSJ[24] := 24;
   // ASSB[18] := 18;
   // ASSB[19] := 19;
   // ASSB[20] := 20;
   // ASSB[21] := 21;
   // ASSB[22] := 22;
   // ASSB[23] := 23;
   // ASSB[24] := 24;
   // PTTS[18] := 20;
   // PTTS[19] := 2;
   // PTTS[20] := 8;
   // PTTS[21] := 12;
   // PTTS[22] := 24;
   // PTTS[23] := 11;
   // PTTS[24] := 25;
   // NTTS[18] := 22;
   // NTTS[19] := 16;
   // NTTS[20] := 24;
   // NTTS[21] := 25;
   // NTTS[22] := 26;
   // NTTS[23] := 27;
   // NTTS[24] := 28;
   // SW_SQTS[18] := 10;
   // SW_SQTS[19] := 1;
   // SW_SQTS[20] := 6;
   // SW_SQTS[21] := 7;
   // SW_SQTS[22] := 6;
   // SW_SQTS[23] := 8;
   // SW_SQTS[24] := 7;
BEGIN
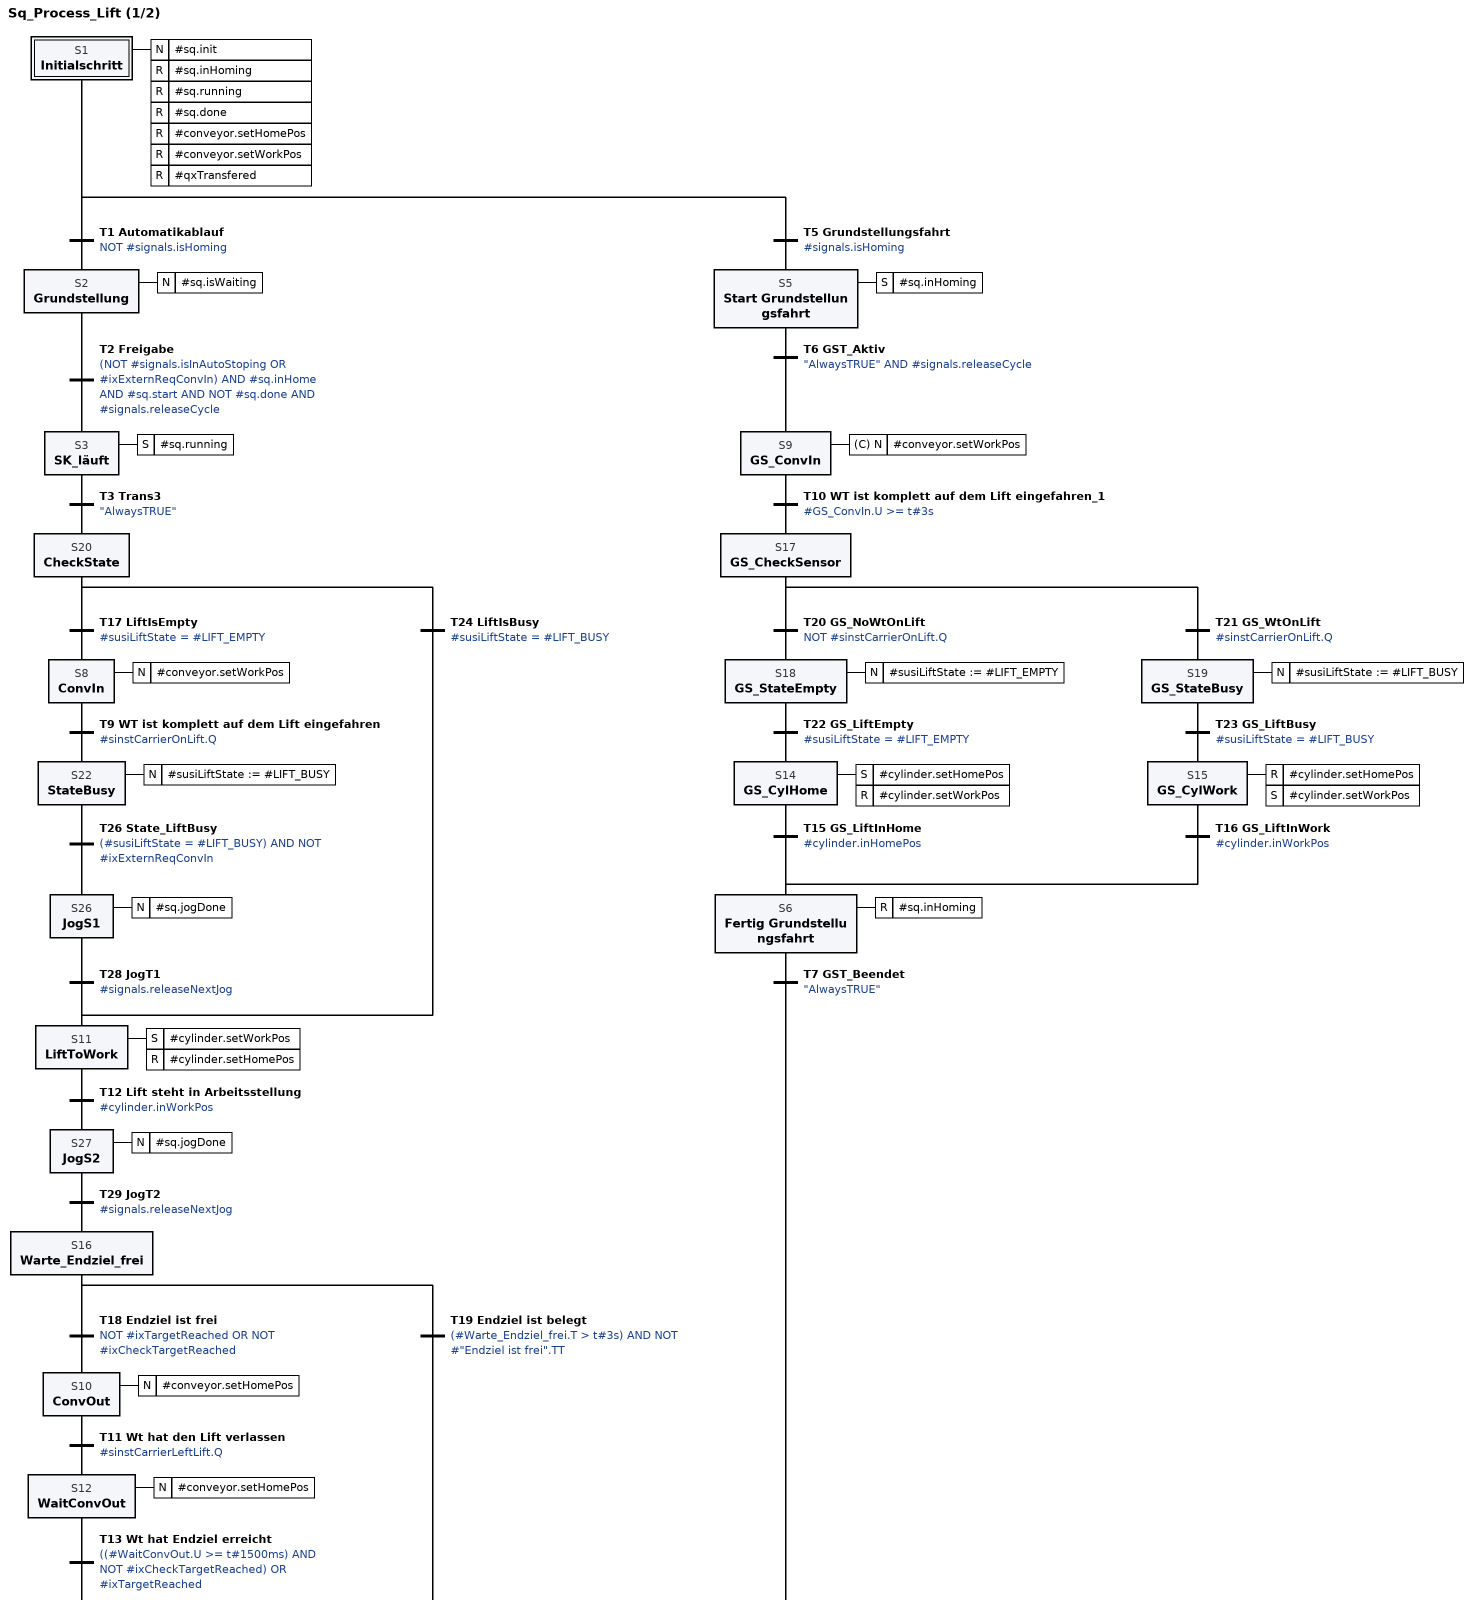
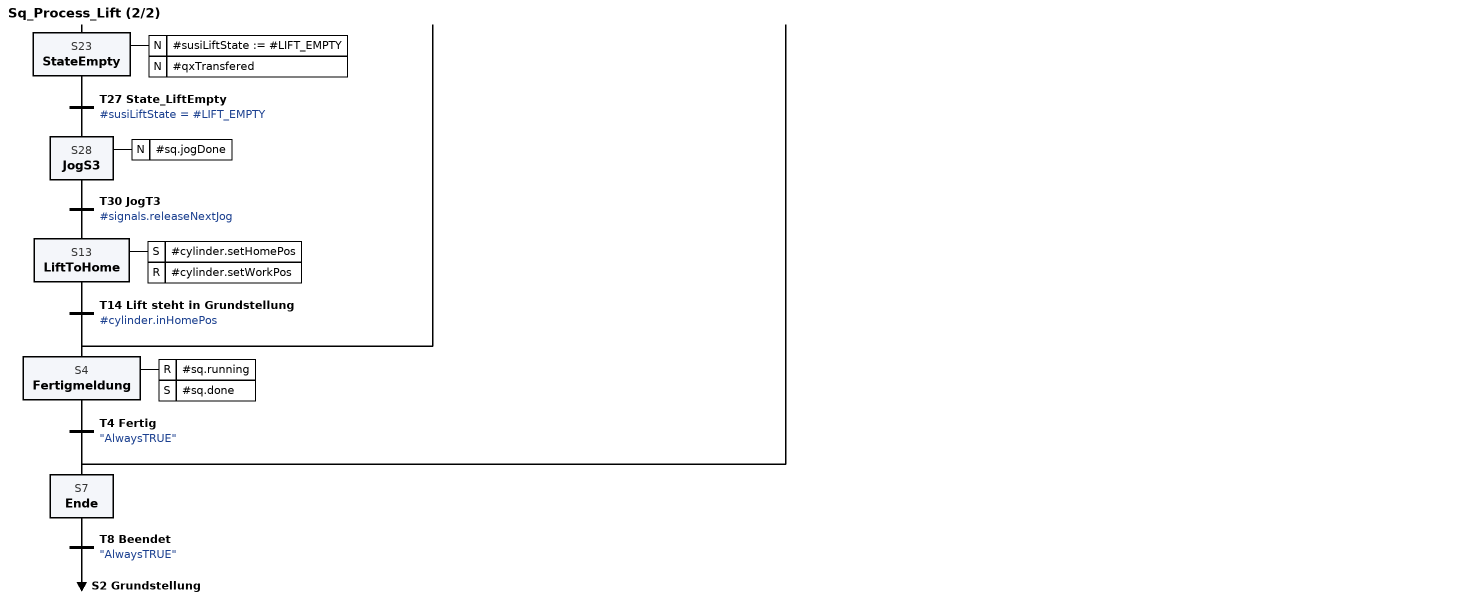
   // permanent pre-instructions
   NETWORK 1
   TITLE = Schrittkette verfügbar / Sequence available
      #sq.exists := true;
   NETWORK 2
   TITLE = WT auf dem Lift / Workpiece carrier on lift
      #sinstCarrierOnLift(IN := #ixCarrierPresent, PT := #itCarrierReactionDelay);   // TON
   NETWORK 3
   TITLE = WT hat Lift verlassen / Workpiece carrier has left lift
      #sinstCarrierLeftLift(IN := NOT #ixCarrierPresent, PT := #itCarrierReactionDelay);   // TON
   NETWORK 4
   TITLE = Schrittkette in Grundstellung (Erweiterbar) / Sequence in home position (extendable)
      #sq.inHome := (((#susiLiftState = #LIFT_EMPTY) AND #cylinder.inHomePos) OR ((#susiLiftState = #LIFT_BUSY) AND #cylinder.inWorkPos)) AND #Grundstellung.X;
   NETWORK 5
   TITLE = Startbedingung (Erweiterbar) / Start condition (extendable)
      #txStartCondition := ((#susiLiftState = #LIFT_EMPTY) AND #ixExternReqConvIn) OR ((#susiLiftState = #LIFT_BUSY) AND (NOT #ixTargetReached OR NOT #ixCheckTargetReached));
   NETWORK 6
   TITLE = Schrittkette starten / Start sequence
      #sq.start := NOT #sq.running AND #signals.releaseCycle AND NOT #signals.isHoming AND #txStartCondition;
      IF #sq.start THEN #sq.done := FALSE; END_IF;
   NETWORK 7
   TITLE = ReleaseCycle-Zeitgeber / ReleaseCycle timer
      // ENO of a box is taken as its EN; it also drops when the box reports an error
      #_w1 := #ERR_FLT AND #ACK_EF;
      #_w2 := #_w1 AND NOT #sstReleaseCycle.ErrorAck;   // rising edge
      #sstReleaseCycle.ErrorAck := #_w1;
      IF (#S_NO <> #sstReleaseCycle.No_LastCycle) OR #_w2 THEN
          #sstReleaseCycle.T := T#0MS;
          #sstReleaseCycle.TckPrev := #sstReleaseCycle.Tck;
          #sstReleaseCycle.No_LastCycle := #S_NO;
      END_IF;
      #sstReleaseCycle.Tck := TIME_TCK();
      #tdTckDiff := #sstReleaseCycle.Tck - #sstReleaseCycle.TckPrev;
      #sstReleaseCycle.TckPrev := #sstReleaseCycle.Tck;
      IF (0 <= #tdTckDiff) AND (#tdTckDiff <= 1000) AND #signals.releaseCycle THEN
          #sstReleaseCycle.T := #sstReleaseCycle.T + #tdTckDiff;
      END_IF;

